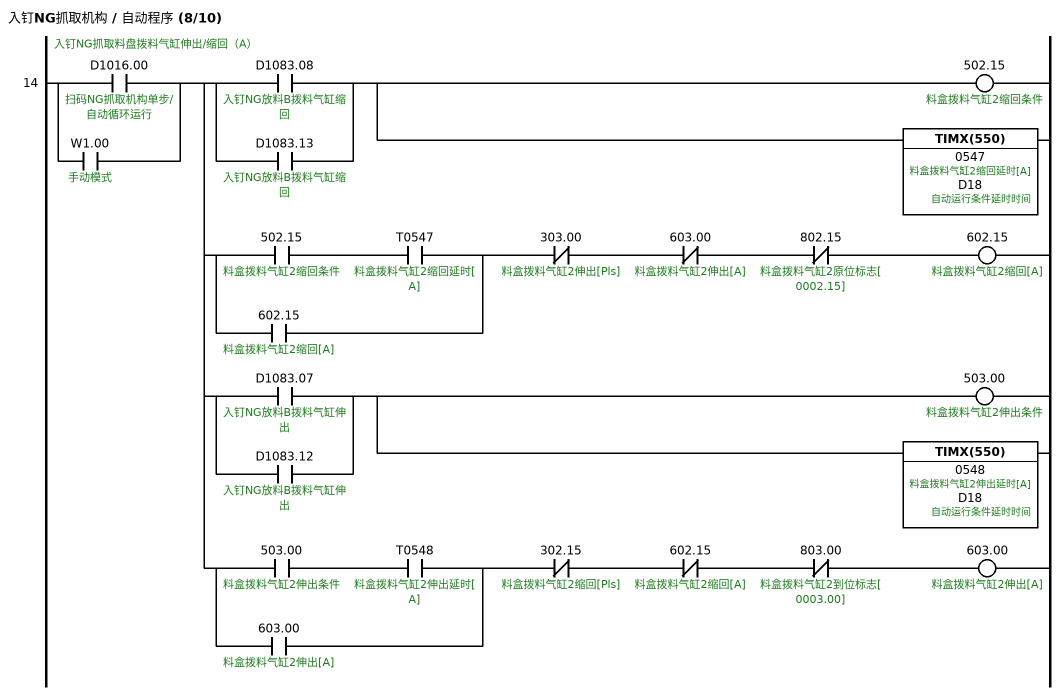
; [picture p144: 入钉NG抓取机构 / 自动程序, rungs 14-14]
; rung 14: 入钉NG抓取料盘拨料气缸伸出/缩回（A）
LD D1016.00  ; 扫码NG抓取机构单步/自动循环运行
OR W1.00  ; 手动模式
OUT TR0
LD D1083.08  ; 入钉NG放料B拨料气缸缩回
OR D1083.13  ; 入钉NG放料B拨料气缸缩回
ANDLD
OUT 502.15  ; 料盒拨料气缸2缩回条件
TIMX(550) 0547 D18  ; 自动运行条件延时时间, 料盒拨料气缸2缩回延时[A]
LD TR0
LD 502.15  ; 料盒拨料气缸2缩回条件
AND T0547  ; 料盒拨料气缸2缩回延时[A]
OR 602.15  ; 料盒拨料气缸2缩回[A]
ANDLD
ANDNOT 303.00  ; 料盒拨料气缸2伸出[Pls]
ANDNOT 603.00  ; 料盒拨料气缸2伸出[A]
ANDNOT 802.15  ; 料盒拨料气缸2原位标志[0002.15]
OUT 602.15  ; 料盒拨料气缸2缩回[A]
LD TR0
LD D1083.07  ; 入钉NG放料B拨料气缸伸出
OR D1083.12  ; 入钉NG放料B拨料气缸伸出
ANDLD
OUT 503.00  ; 料盒拨料气缸2伸出条件
TIMX(550) 0548 D18  ; 自动运行条件延时时间, 料盒拨料气缸2伸出延时[A]
LD TR0
LD 503.00  ; 料盒拨料气缸2伸出条件
AND T0548  ; 料盒拨料气缸2伸出延时[A]
OR 603.00  ; 料盒拨料气缸2伸出[A]
ANDLD
ANDNOT 302.15  ; 料盒拨料气缸2缩回[Pls]
ANDNOT 602.15  ; 料盒拨料气缸2缩回[A]
ANDNOT 803.00  ; 料盒拨料气缸2到位标志[0003.00]
OUT 603.00  ; 料盒拨料气缸2伸出[A]

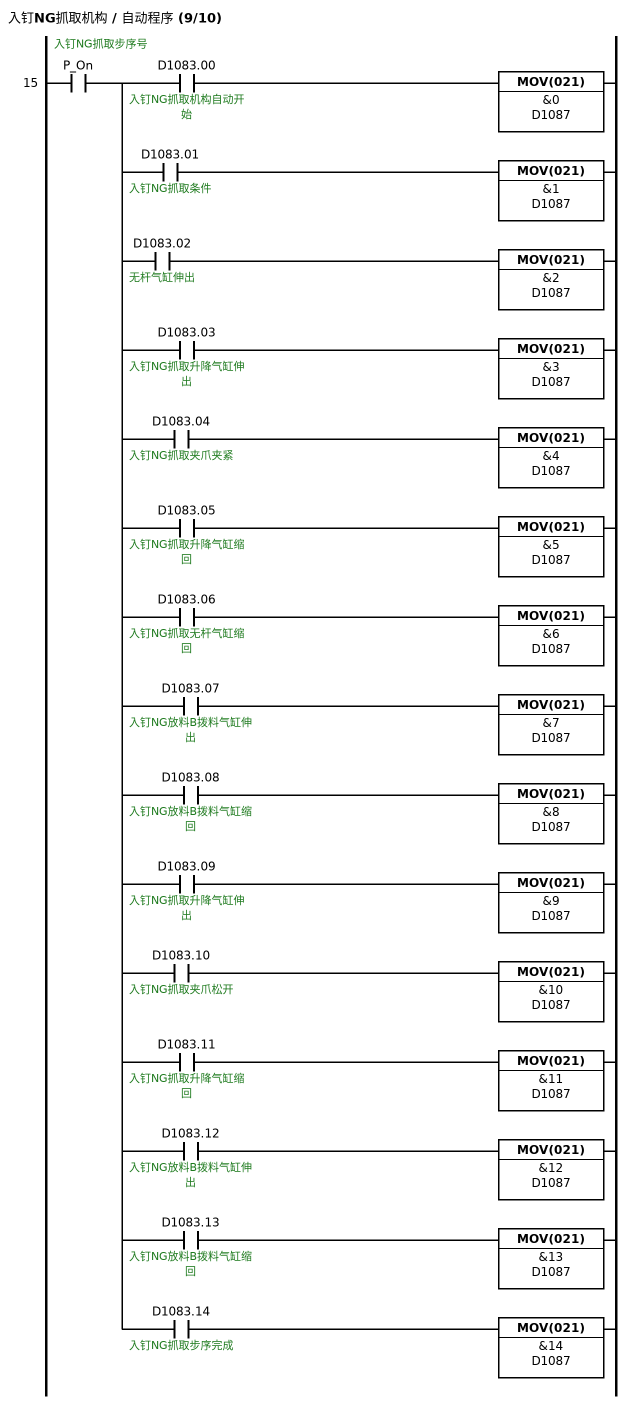
; rung 15: 入钉NG抓取步序号
LD P_On
OUT TR0
AND D1083.00  ; 入钉NG抓取机构自动开始
MOV(021) &0 D1087
LD TR0
AND D1083.01  ; 入钉NG抓取条件
MOV(021) &1 D1087
LD TR0
AND D1083.02  ; 无杆气缸伸出
MOV(021) &2 D1087
LD TR0
AND D1083.03  ; 入钉NG抓取升降气缸伸出
MOV(021) &3 D1087
LD TR0
AND D1083.04  ; 入钉NG抓取夹爪夹紧
MOV(021) &4 D1087
LD TR0
AND D1083.05  ; 入钉NG抓取升降气缸缩回
MOV(021) &5 D1087
LD TR0
AND D1083.06  ; 入钉NG抓取无杆气缸缩回
MOV(021) &6 D1087
LD TR0
AND D1083.07  ; 入钉NG放料B拨料气缸伸出
MOV(021) &7 D1087
LD TR0
AND D1083.08  ; 入钉NG放料B拨料气缸缩回
MOV(021) &8 D1087
LD TR0
AND D1083.09  ; 入钉NG抓取升降气缸伸出
MOV(021) &9 D1087
LD TR0
AND D1083.10  ; 入钉NG抓取夹爪松开
MOV(021) &10 D1087
LD TR0
AND D1083.11  ; 入钉NG抓取升降气缸缩回
MOV(021) &11 D1087
LD TR0
AND D1083.12  ; 入钉NG放料B拨料气缸伸出
MOV(021) &12 D1087
LD TR0
AND D1083.13  ; 入钉NG放料B拨料气缸缩回
MOV(021) &13 D1087
LD TR0
AND D1083.14  ; 入钉NG抓取步序完成
MOV(021) &14 D1087

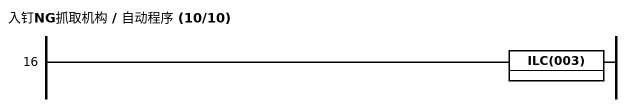
; rung 16
ILC(003)

### Section 状态指示灯

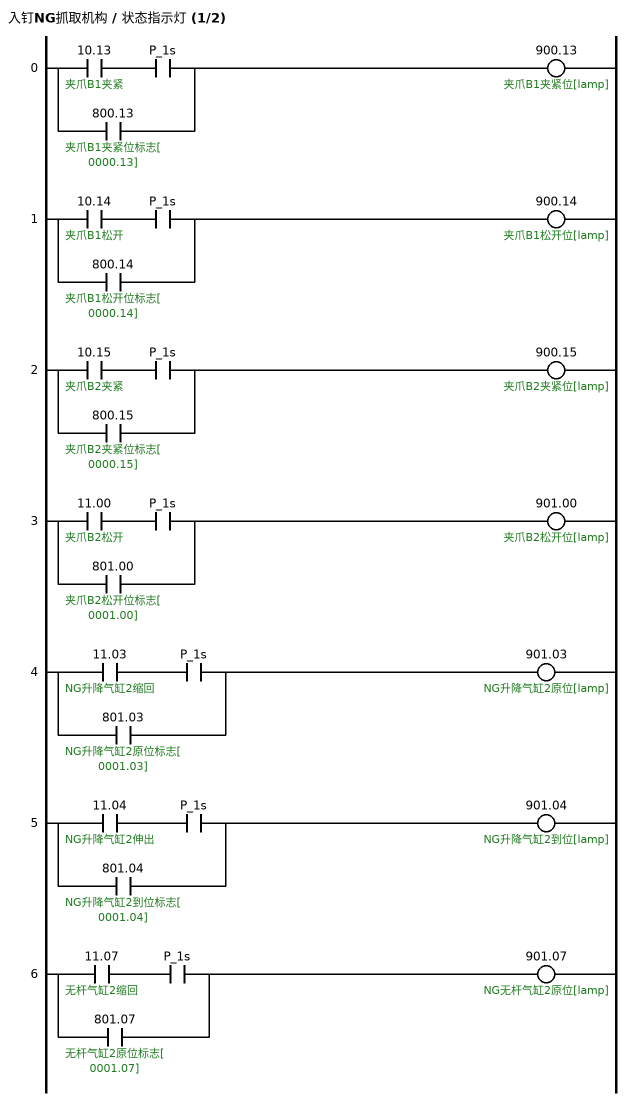
; rung 0
LD 10.13  ; 夹爪B1夹紧
AND P_1s
OR 800.13  ; 夹爪B1夹紧位标志[0000.13]
OUT 900.13  ; 夹爪B1夹紧位[lamp]
; rung 1
LD 10.14  ; 夹爪B1松开
AND P_1s
OR 800.14  ; 夹爪B1松开位标志[0000.14]
OUT 900.14  ; 夹爪B1松开位[lamp]
; rung 2
LD 10.15  ; 夹爪B2夹紧
AND P_1s
OR 800.15  ; 夹爪B2夹紧位标志[0000.15]
OUT 900.15  ; 夹爪B2夹紧位[lamp]
; rung 3
LD 11.00  ; 夹爪B2松开
AND P_1s
OR 801.00  ; 夹爪B2松开位标志[0001.00]
OUT 901.00  ; 夹爪B2松开位[lamp]
; rung 4
LD 11.03  ; NG升降气缸2缩回
AND P_1s
OR 801.03  ; NG升降气缸2原位标志[0001.03]
OUT 901.03  ; NG升降气缸2原位[lamp]
; rung 5
LD 11.04  ; NG升降气缸2伸出
AND P_1s
OR 801.04  ; NG升降气缸2到位标志[0001.04]
OUT 901.04  ; NG升降气缸2到位[lamp]
; rung 6
LD 11.07  ; 无杆气缸2缩回
AND P_1s
OR 801.07  ; 无杆气缸2原位标志[0001.07]
OUT 901.07  ; NG无杆气缸2原位[lamp]

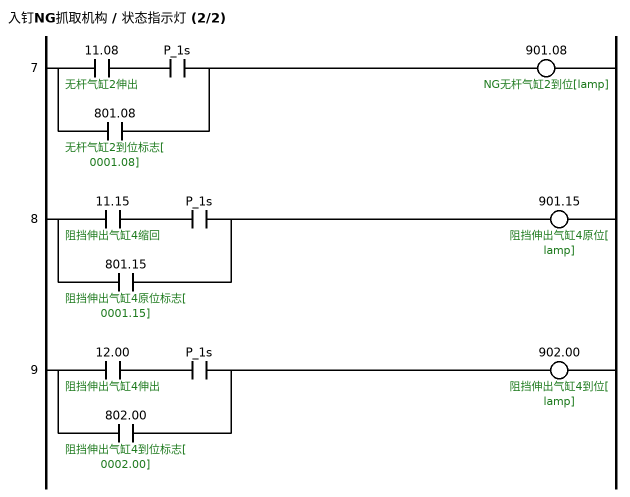
; rung 7
LD 11.08  ; 无杆气缸2伸出
AND P_1s
OR 801.08  ; 无杆气缸2到位标志[0001.08]
OUT 901.08  ; NG无杆气缸2到位[lamp]
; rung 8
LD 11.15  ; 阻挡伸出气缸4缩回
AND P_1s
OR 801.15  ; 阻挡伸出气缸4原位标志[0001.15]
OUT 901.15  ; 阻挡伸出气缸4原位[lamp]
; rung 9
LD 12.00  ; 阻挡伸出气缸4伸出
AND P_1s
OR 802.00  ; 阻挡伸出气缸4到位标志[0002.00]
OUT 902.00  ; 阻挡伸出气缸4到位[lamp]

### Section 输出程序

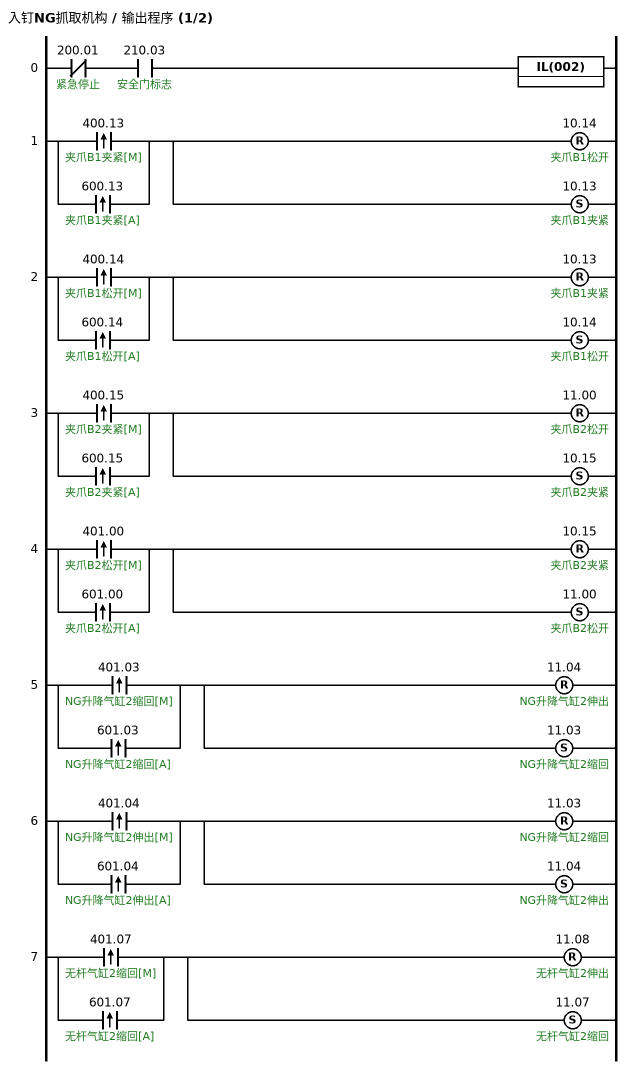
; rung 0
LDNOT 200.01  ; 紧急停止
AND 210.03  ; 安全门标志
IL(002)
; rung 1
@LD 400.13  ; 夹爪B1夹紧[M]
@OR 600.13  ; 夹爪B1夹紧[A]
RSET 10.14  ; 夹爪B1松开
SET 10.13  ; 夹爪B1夹紧
; rung 2
@LD 400.14  ; 夹爪B1松开[M]
@OR 600.14  ; 夹爪B1松开[A]
RSET 10.13  ; 夹爪B1夹紧
SET 10.14  ; 夹爪B1松开
; rung 3
@LD 400.15  ; 夹爪B2夹紧[M]
@OR 600.15  ; 夹爪B2夹紧[A]
RSET 11.00  ; 夹爪B2松开
SET 10.15  ; 夹爪B2夹紧
; rung 4
@LD 401.00  ; 夹爪B2松开[M]
@OR 601.00  ; 夹爪B2松开[A]
RSET 10.15  ; 夹爪B2夹紧
SET 11.00  ; 夹爪B2松开
; rung 5
@LD 401.03  ; NG升降气缸2缩回[M]
@OR 601.03  ; NG升降气缸2缩回[A]
RSET 11.04  ; NG升降气缸2伸出
SET 11.03  ; NG升降气缸2缩回
; rung 6
@LD 401.04  ; NG升降气缸2伸出[M]
@OR 601.04  ; NG升降气缸2伸出[A]
RSET 11.03  ; NG升降气缸2缩回
SET 11.04  ; NG升降气缸2伸出
; rung 7
@LD 401.07  ; 无杆气缸2缩回[M]
@OR 601.07  ; 无杆气缸2缩回[A]
RSET 11.08  ; 无杆气缸2伸出
SET 11.07  ; 无杆气缸2缩回

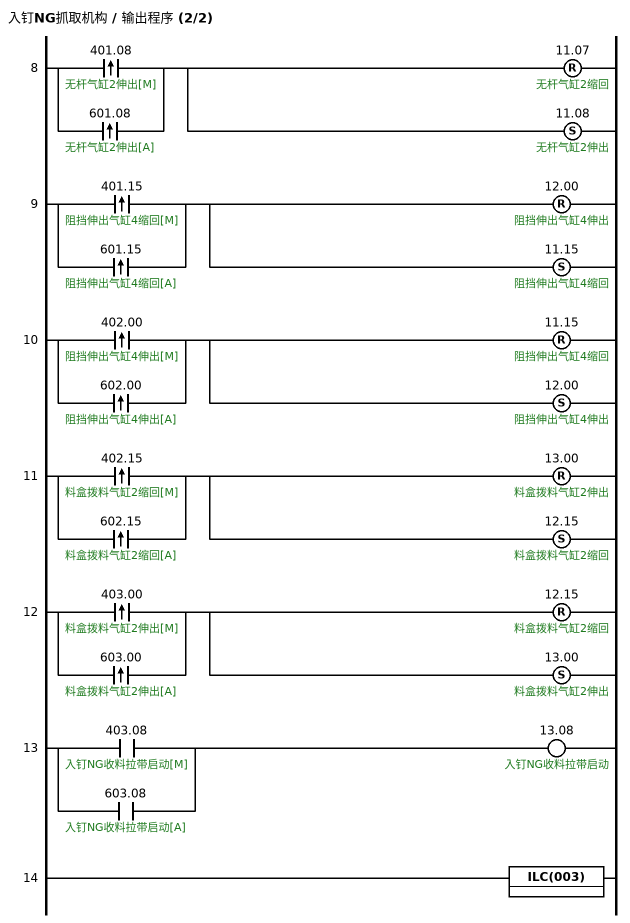
; rung 8
@LD 401.08  ; 无杆气缸2伸出[M]
@OR 601.08  ; 无杆气缸2伸出[A]
RSET 11.07  ; 无杆气缸2缩回
SET 11.08  ; 无杆气缸2伸出
; rung 9
@LD 401.15  ; 阻挡伸出气缸4缩回[M]
@OR 601.15  ; 阻挡伸出气缸4缩回[A]
RSET 12.00  ; 阻挡伸出气缸4伸出
SET 11.15  ; 阻挡伸出气缸4缩回
; rung 10
@LD 402.00  ; 阻挡伸出气缸4伸出[M]
@OR 602.00  ; 阻挡伸出气缸4伸出[A]
RSET 11.15  ; 阻挡伸出气缸4缩回
SET 12.00  ; 阻挡伸出气缸4伸出
; rung 11
@LD 402.15  ; 料盒拨料气缸2缩回[M]
@OR 602.15  ; 料盒拨料气缸2缩回[A]
RSET 13.00  ; 料盒拨料气缸2伸出
SET 12.15  ; 料盒拨料气缸2缩回
; rung 12
@LD 403.00  ; 料盒拨料气缸2伸出[M]
@OR 603.00  ; 料盒拨料气缸2伸出[A]
RSET 12.15  ; 料盒拨料气缸2缩回
SET 13.00  ; 料盒拨料气缸2伸出
; rung 13
LD 403.08  ; 入钉NG收料拉带启动[M]
OR 603.08  ; 入钉NG收料拉带启动[A]
OUT 13.08  ; 入钉NG收料拉带启动
; rung 14
ILC(003)

### Section END
; rung 0
END(001)

## Program COMMON (cyclic task 6)

### Section 传感器延时

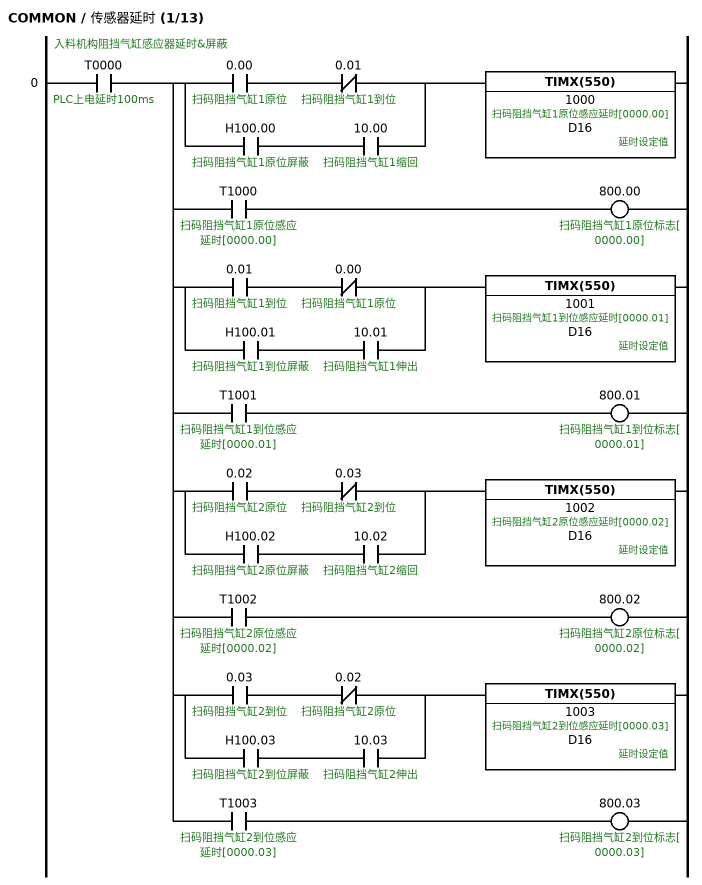
; rung 0: 入料机构阻挡气缸感应器延时&屏蔽
LD T0000  ; PLC上电延时100ms
OUT TR0
LD 0.00  ; 扫码阻挡气缸1原位
ANDNOT 0.01  ; 扫码阻挡气缸1到位
LD H100.00  ; 扫码阻挡气缸1原位屏蔽
AND 10.00  ; 扫码阻挡气缸1缩回
ORLD
ANDLD
TIMX(550) 1000 D16  ; 延时设定值, 扫码阻挡气缸1原位感应延时[0000.00]
LD TR0
AND T1000  ; 扫码阻挡气缸1原位感应延时[0000.00]
OUT 800.00  ; 扫码阻挡气缸1原位标志[0000.00]
LD TR0
LD 0.01  ; 扫码阻挡气缸1到位
ANDNOT 0.00  ; 扫码阻挡气缸1原位
LD H100.01  ; 扫码阻挡气缸1到位屏蔽
AND 10.01  ; 扫码阻挡气缸1伸出
ORLD
ANDLD
TIMX(550) 1001 D16  ; 延时设定值, 扫码阻挡气缸1到位感应延时[0000.01]
LD TR0
AND T1001  ; 扫码阻挡气缸1到位感应延时[0000.01]
OUT 800.01  ; 扫码阻挡气缸1到位标志[0000.01]
LD TR0
LD 0.02  ; 扫码阻挡气缸2原位
ANDNOT 0.03  ; 扫码阻挡气缸2到位
LD H100.02  ; 扫码阻挡气缸2原位屏蔽
AND 10.02  ; 扫码阻挡气缸2缩回
ORLD
ANDLD
TIMX(550) 1002 D16  ; 延时设定值, 扫码阻挡气缸2原位感应延时[0000.02]
LD TR0
AND T1002  ; 扫码阻挡气缸2原位感应延时[0000.02]
OUT 800.02  ; 扫码阻挡气缸2原位标志[0000.02]
LD TR0
LD 0.03  ; 扫码阻挡气缸2到位
ANDNOT 0.02  ; 扫码阻挡气缸2原位
LD H100.03  ; 扫码阻挡气缸2到位屏蔽
AND 10.03  ; 扫码阻挡气缸2伸出
ORLD
ANDLD
TIMX(550) 1003 D16  ; 延时设定值, 扫码阻挡气缸2到位感应延时[0000.03]
LD TR0
AND T1003  ; 扫码阻挡气缸2到位感应延时[0000.03]
OUT 800.03  ; 扫码阻挡气缸2到位标志[0000.03]

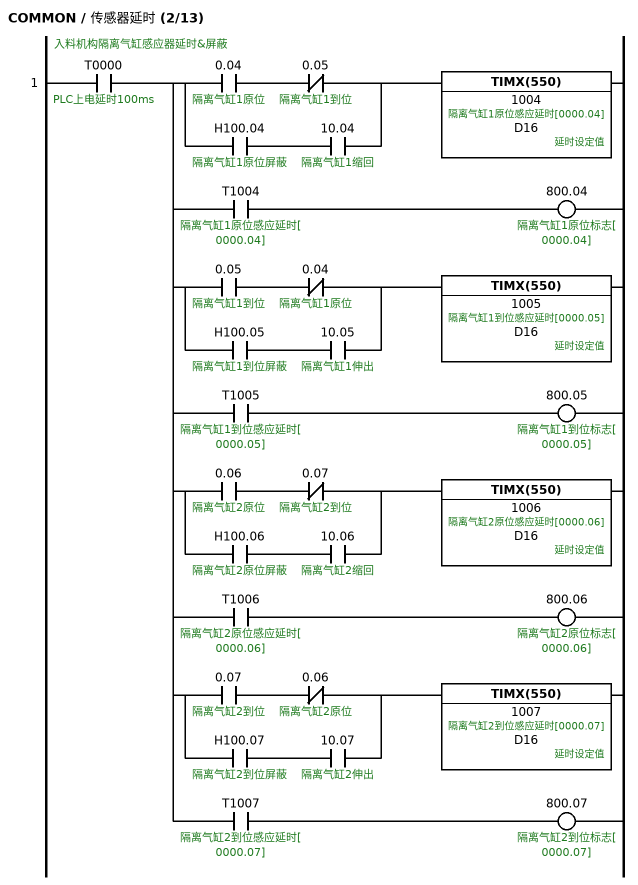
; rung 1: 入料机构隔离气缸感应器延时&屏蔽
LD T0000  ; PLC上电延时100ms
OUT TR0
LD 0.04  ; 隔离气缸1原位
ANDNOT 0.05  ; 隔离气缸1到位
LD H100.04  ; 隔离气缸1原位屏蔽
AND 10.04  ; 隔离气缸1缩回
ORLD
ANDLD
TIMX(550) 1004 D16  ; 延时设定值, 隔离气缸1原位感应延时[0000.04]
LD TR0
AND T1004  ; 隔离气缸1原位感应延时[0000.04]
OUT 800.04  ; 隔离气缸1原位标志[0000.04]
LD TR0
LD 0.05  ; 隔离气缸1到位
ANDNOT 0.04  ; 隔离气缸1原位
LD H100.05  ; 隔离气缸1到位屏蔽
AND 10.05  ; 隔离气缸1伸出
ORLD
ANDLD
TIMX(550) 1005 D16  ; 延时设定值, 隔离气缸1到位感应延时[0000.05]
LD TR0
AND T1005  ; 隔离气缸1到位感应延时[0000.05]
OUT 800.05  ; 隔离气缸1到位标志[0000.05]
LD TR0
LD 0.06  ; 隔离气缸2原位
ANDNOT 0.07  ; 隔离气缸2到位
LD H100.06  ; 隔离气缸2原位屏蔽
AND 10.06  ; 隔离气缸2缩回
ORLD
ANDLD
TIMX(550) 1006 D16  ; 延时设定值, 隔离气缸2原位感应延时[0000.06]
LD TR0
AND T1006  ; 隔离气缸2原位感应延时[0000.06]
OUT 800.06  ; 隔离气缸2原位标志[0000.06]
LD TR0
LD 0.07  ; 隔离气缸2到位
ANDNOT 0.06  ; 隔离气缸2原位
LD H100.07  ; 隔离气缸2到位屏蔽
AND 10.07  ; 隔离气缸2伸出
ORLD
ANDLD
TIMX(550) 1007 D16  ; 延时设定值, 隔离气缸2到位感应延时[0000.07]
LD TR0
AND T1007  ; 隔离气缸2到位感应延时[0000.07]
OUT 800.07  ; 隔离气缸2到位标志[0000.07]

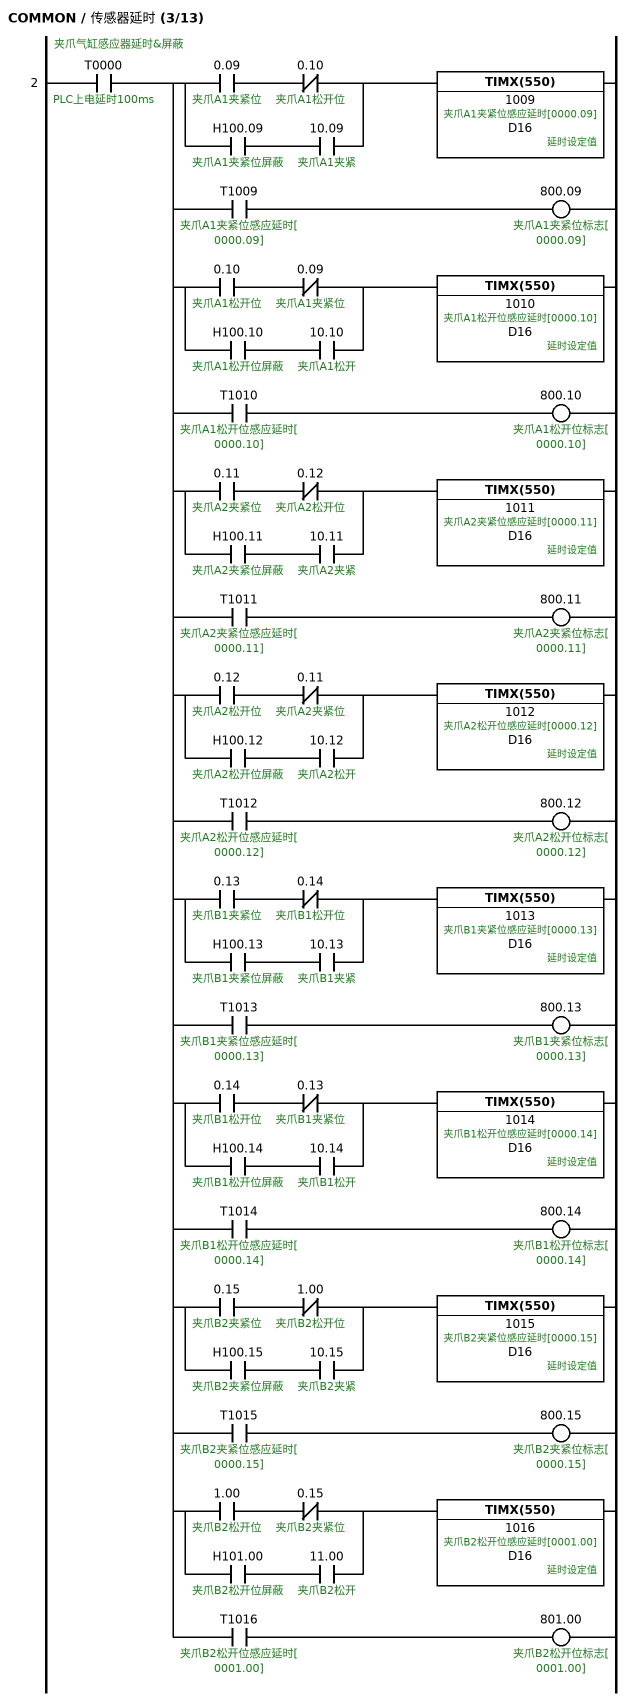
; rung 2: 夹爪气缸感应器延时&屏蔽
LD T0000  ; PLC上电延时100ms
OUT TR0
LD 0.09  ; 夹爪A1夹紧位
ANDNOT 0.10  ; 夹爪A1松开位
LD H100.09  ; 夹爪A1夹紧位屏蔽
AND 10.09  ; 夹爪A1夹紧
ORLD
ANDLD
TIMX(550) 1009 D16  ; 延时设定值, 夹爪A1夹紧位感应延时[0000.09]
LD TR0
AND T1009  ; 夹爪A1夹紧位感应延时[0000.09]
OUT 800.09  ; 夹爪A1夹紧位标志[0000.09]
LD TR0
LD 0.10  ; 夹爪A1松开位
ANDNOT 0.09  ; 夹爪A1夹紧位
LD H100.10  ; 夹爪A1松开位屏蔽
AND 10.10  ; 夹爪A1松开
ORLD
ANDLD
TIMX(550) 1010 D16  ; 延时设定值, 夹爪A1松开位感应延时[0000.10]
LD TR0
AND T1010  ; 夹爪A1松开位感应延时[0000.10]
OUT 800.10  ; 夹爪A1松开位标志[0000.10]
LD TR0
LD 0.11  ; 夹爪A2夹紧位
ANDNOT 0.12  ; 夹爪A2松开位
LD H100.11  ; 夹爪A2夹紧位屏蔽
AND 10.11  ; 夹爪A2夹紧
ORLD
ANDLD
TIMX(550) 1011 D16  ; 延时设定值, 夹爪A2夹紧位感应延时[0000.11]
LD TR0
AND T1011  ; 夹爪A2夹紧位感应延时[0000.11]
OUT 800.11  ; 夹爪A2夹紧位标志[0000.11]
LD TR0
LD 0.12  ; 夹爪A2松开位
ANDNOT 0.11  ; 夹爪A2夹紧位
LD H100.12  ; 夹爪A2松开位屏蔽
AND 10.12  ; 夹爪A2松开
ORLD
ANDLD
TIMX(550) 1012 D16  ; 延时设定值, 夹爪A2松开位感应延时[0000.12]
LD TR0
AND T1012  ; 夹爪A2松开位感应延时[0000.12]
OUT 800.12  ; 夹爪A2松开位标志[0000.12]
LD TR0
LD 0.13  ; 夹爪B1夹紧位
ANDNOT 0.14  ; 夹爪B1松开位
LD H100.13  ; 夹爪B1夹紧位屏蔽
AND 10.13  ; 夹爪B1夹紧
ORLD
ANDLD
TIMX(550) 1013 D16  ; 延时设定值, 夹爪B1夹紧位感应延时[0000.13]
LD TR0
AND T1013  ; 夹爪B1夹紧位感应延时[0000.13]
OUT 800.13  ; 夹爪B1夹紧位标志[0000.13]
LD TR0
LD 0.14  ; 夹爪B1松开位
ANDNOT 0.13  ; 夹爪B1夹紧位
LD H100.14  ; 夹爪B1松开位屏蔽
AND 10.14  ; 夹爪B1松开
ORLD
ANDLD
TIMX(550) 1014 D16  ; 延时设定值, 夹爪B1松开位感应延时[0000.14]
LD TR0
AND T1014  ; 夹爪B1松开位感应延时[0000.14]
OUT 800.14  ; 夹爪B1松开位标志[0000.14]
LD TR0
LD 0.15  ; 夹爪B2夹紧位
ANDNOT 1.00  ; 夹爪B2松开位
LD H100.15  ; 夹爪B2夹紧位屏蔽
AND 10.15  ; 夹爪B2夹紧
ORLD
ANDLD
TIMX(550) 1015 D16  ; 延时设定值, 夹爪B2夹紧位感应延时[0000.15]
LD TR0
AND T1015  ; 夹爪B2夹紧位感应延时[0000.15]
OUT 800.15  ; 夹爪B2夹紧位标志[0000.15]
LD TR0
LD 1.00  ; 夹爪B2松开位
ANDNOT 0.15  ; 夹爪B2夹紧位
LD H101.00  ; 夹爪B2松开位屏蔽
AND 11.00  ; 夹爪B2松开
ORLD
ANDLD
TIMX(550) 1016 D16  ; 延时设定值, 夹爪B2松开位感应延时[0001.00]
LD TR0
AND T1016  ; 夹爪B2松开位感应延时[0001.00]
OUT 801.00  ; 夹爪B2松开位标志[0001.00]

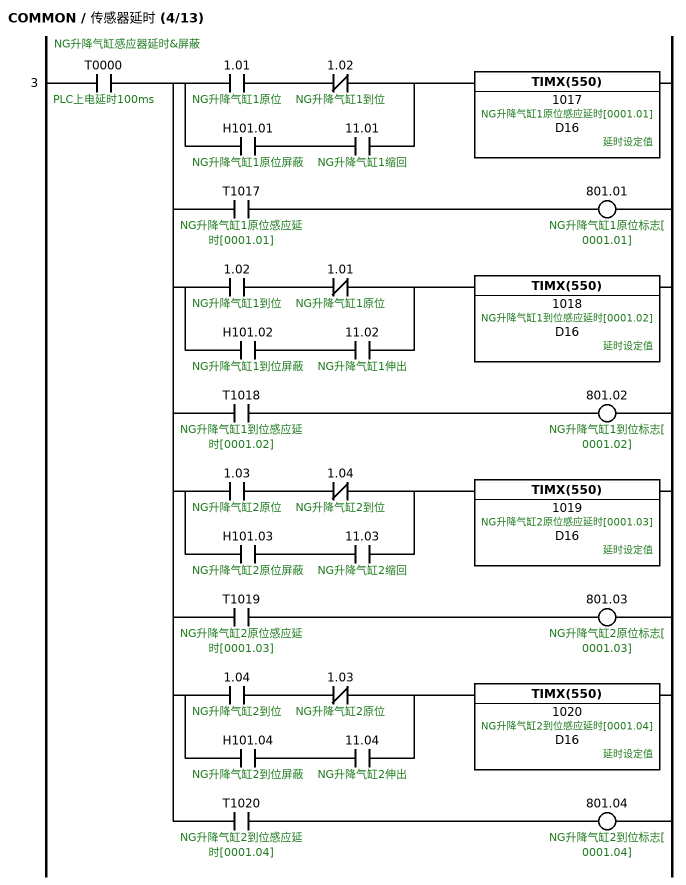
; rung 3: NG升降气缸感应器延时&屏蔽
LD T0000  ; PLC上电延时100ms
OUT TR0
LD 1.01  ; NG升降气缸1原位
ANDNOT 1.02  ; NG升降气缸1到位
LD H101.01  ; NG升降气缸1原位屏蔽
AND 11.01  ; NG升降气缸1缩回
ORLD
ANDLD
TIMX(550) 1017 D16  ; 延时设定值, NG升降气缸1原位感应延时[0001.01]
LD TR0
AND T1017  ; NG升降气缸1原位感应延时[0001.01]
OUT 801.01  ; NG升降气缸1原位标志[0001.01]
LD TR0
LD 1.02  ; NG升降气缸1到位
ANDNOT 1.01  ; NG升降气缸1原位
LD H101.02  ; NG升降气缸1到位屏蔽
AND 11.02  ; NG升降气缸1伸出
ORLD
ANDLD
TIMX(550) 1018 D16  ; 延时设定值, NG升降气缸1到位感应延时[0001.02]
LD TR0
AND T1018  ; NG升降气缸1到位感应延时[0001.02]
OUT 801.02  ; NG升降气缸1到位标志[0001.02]
LD TR0
LD 1.03  ; NG升降气缸2原位
ANDNOT 1.04  ; NG升降气缸2到位
LD H101.03  ; NG升降气缸2原位屏蔽
AND 11.03  ; NG升降气缸2缩回
ORLD
ANDLD
TIMX(550) 1019 D16  ; 延时设定值, NG升降气缸2原位感应延时[0001.03]
LD TR0
AND T1019  ; NG升降气缸2原位感应延时[0001.03]
OUT 801.03  ; NG升降气缸2原位标志[0001.03]
LD TR0
LD 1.04  ; NG升降气缸2到位
ANDNOT 1.03  ; NG升降气缸2原位
LD H101.04  ; NG升降气缸2到位屏蔽
AND 11.04  ; NG升降气缸2伸出
ORLD
ANDLD
TIMX(550) 1020 D16  ; 延时设定值, NG升降气缸2到位感应延时[0001.04]
LD TR0
AND T1020  ; NG升降气缸2到位感应延时[0001.04]
OUT 801.04  ; NG升降气缸2到位标志[0001.04]

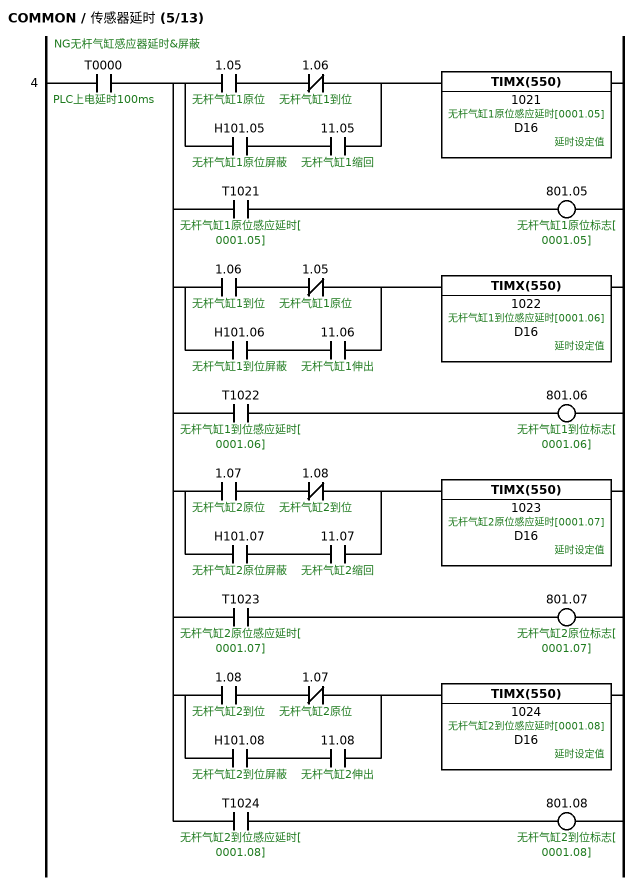
; rung 4: NG无杆气缸感应器延时&屏蔽
LD T0000  ; PLC上电延时100ms
OUT TR0
LD 1.05  ; 无杆气缸1原位
ANDNOT 1.06  ; 无杆气缸1到位
LD H101.05  ; 无杆气缸1原位屏蔽
AND 11.05  ; 无杆气缸1缩回
ORLD
ANDLD
TIMX(550) 1021 D16  ; 延时设定值, 无杆气缸1原位感应延时[0001.05]
LD TR0
AND T1021  ; 无杆气缸1原位感应延时[0001.05]
OUT 801.05  ; 无杆气缸1原位标志[0001.05]
LD TR0
LD 1.06  ; 无杆气缸1到位
ANDNOT 1.05  ; 无杆气缸1原位
LD H101.06  ; 无杆气缸1到位屏蔽
AND 11.06  ; 无杆气缸1伸出
ORLD
ANDLD
TIMX(550) 1022 D16  ; 延时设定值, 无杆气缸1到位感应延时[0001.06]
LD TR0
AND T1022  ; 无杆气缸1到位感应延时[0001.06]
OUT 801.06  ; 无杆气缸1到位标志[0001.06]
LD TR0
LD 1.07  ; 无杆气缸2原位
ANDNOT 1.08  ; 无杆气缸2到位
LD H101.07  ; 无杆气缸2原位屏蔽
AND 11.07  ; 无杆气缸2缩回
ORLD
ANDLD
TIMX(550) 1023 D16  ; 延时设定值, 无杆气缸2原位感应延时[0001.07]
LD TR0
AND T1023  ; 无杆气缸2原位感应延时[0001.07]
OUT 801.07  ; 无杆气缸2原位标志[0001.07]
LD TR0
LD 1.08  ; 无杆气缸2到位
ANDNOT 1.07  ; 无杆气缸2原位
LD H101.08  ; 无杆气缸2到位屏蔽
AND 11.08  ; 无杆气缸2伸出
ORLD
ANDLD
TIMX(550) 1024 D16  ; 延时设定值, 无杆气缸2到位感应延时[0001.08]
LD TR0
AND T1024  ; 无杆气缸2到位感应延时[0001.08]
OUT 801.08  ; 无杆气缸2到位标志[0001.08]

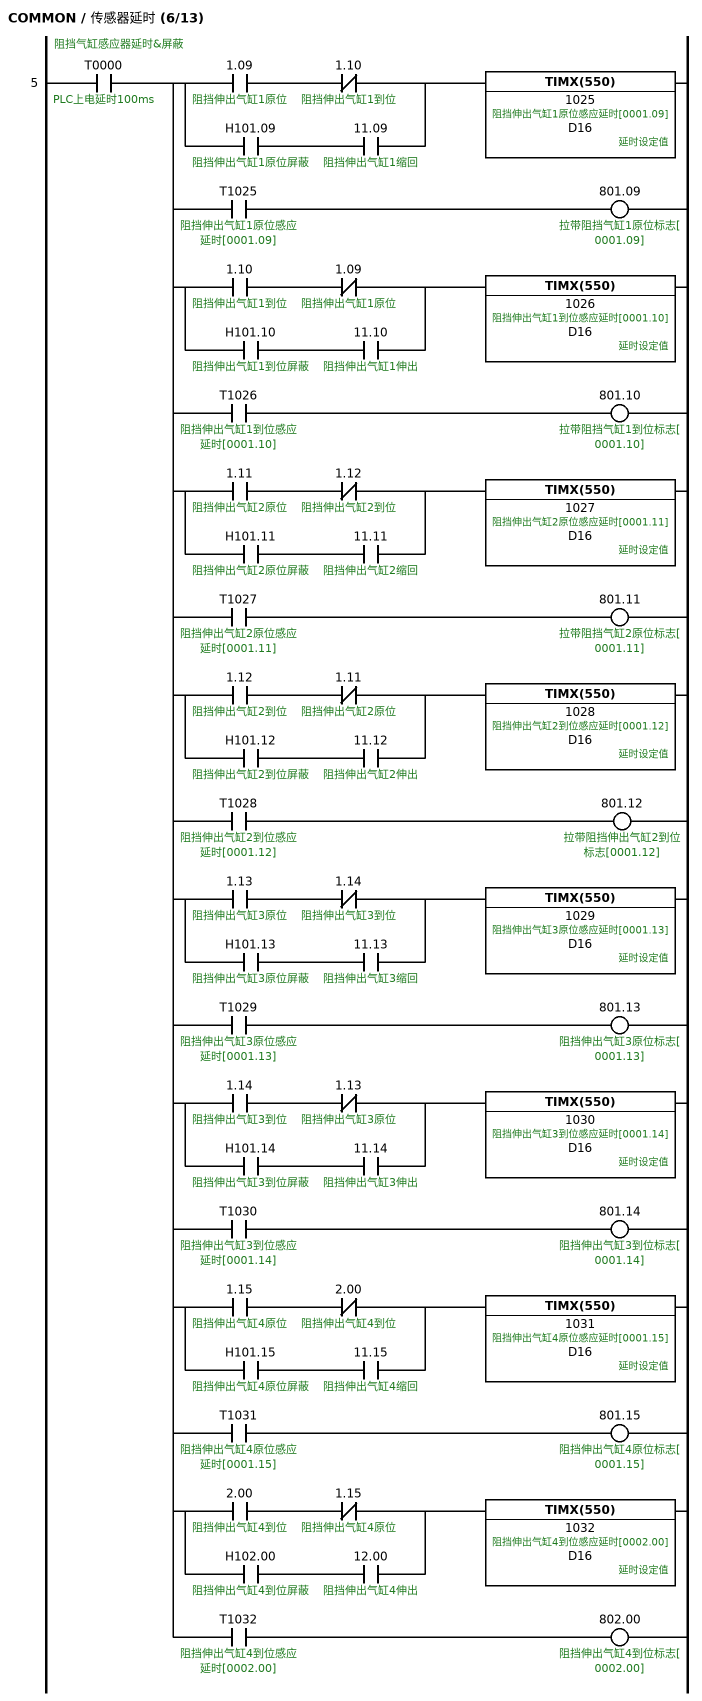
; rung 5: 阻挡气缸感应器延时&屏蔽
LD T0000  ; PLC上电延时100ms
OUT TR0
LD 1.09  ; 阻挡伸出气缸1原位
ANDNOT 1.10  ; 阻挡伸出气缸1到位
LD H101.09  ; 阻挡伸出气缸1原位屏蔽
AND 11.09  ; 阻挡伸出气缸1缩回
ORLD
ANDLD
TIMX(550) 1025 D16  ; 延时设定值, 阻挡伸出气缸1原位感应延时[0001.09]
LD TR0
AND T1025  ; 阻挡伸出气缸1原位感应延时[0001.09]
OUT 801.09  ; 拉带阻挡气缸1原位标志[0001.09]
LD TR0
LD 1.10  ; 阻挡伸出气缸1到位
ANDNOT 1.09  ; 阻挡伸出气缸1原位
LD H101.10  ; 阻挡伸出气缸1到位屏蔽
AND 11.10  ; 阻挡伸出气缸1伸出
ORLD
ANDLD
TIMX(550) 1026 D16  ; 延时设定值, 阻挡伸出气缸1到位感应延时[0001.10]
LD TR0
AND T1026  ; 阻挡伸出气缸1到位感应延时[0001.10]
OUT 801.10  ; 拉带阻挡气缸1到位标志[0001.10]
LD TR0
LD 1.11  ; 阻挡伸出气缸2原位
ANDNOT 1.12  ; 阻挡伸出气缸2到位
LD H101.11  ; 阻挡伸出气缸2原位屏蔽
AND 11.11  ; 阻挡伸出气缸2缩回
ORLD
ANDLD
TIMX(550) 1027 D16  ; 延时设定值, 阻挡伸出气缸2原位感应延时[0001.11]
LD TR0
AND T1027  ; 阻挡伸出气缸2原位感应延时[0001.11]
OUT 801.11  ; 拉带阻挡气缸2原位标志[0001.11]
LD TR0
LD 1.12  ; 阻挡伸出气缸2到位
ANDNOT 1.11  ; 阻挡伸出气缸2原位
LD H101.12  ; 阻挡伸出气缸2到位屏蔽
AND 11.12  ; 阻挡伸出气缸2伸出
ORLD
ANDLD
TIMX(550) 1028 D16  ; 延时设定值, 阻挡伸出气缸2到位感应延时[0001.12]
LD TR0
AND T1028  ; 阻挡伸出气缸2到位感应延时[0001.12]
OUT 801.12  ; 拉带阻挡伸出气缸2到位标志[0001.12]
LD TR0
LD 1.13  ; 阻挡伸出气缸3原位
ANDNOT 1.14  ; 阻挡伸出气缸3到位
LD H101.13  ; 阻挡伸出气缸3原位屏蔽
AND 11.13  ; 阻挡伸出气缸3缩回
ORLD
ANDLD
TIMX(550) 1029 D16  ; 延时设定值, 阻挡伸出气缸3原位感应延时[0001.13]
LD TR0
AND T1029  ; 阻挡伸出气缸3原位感应延时[0001.13]
OUT 801.13  ; 阻挡伸出气缸3原位标志[0001.13]
LD TR0
LD 1.14  ; 阻挡伸出气缸3到位
ANDNOT 1.13  ; 阻挡伸出气缸3原位
LD H101.14  ; 阻挡伸出气缸3到位屏蔽
AND 11.14  ; 阻挡伸出气缸3伸出
ORLD
ANDLD
TIMX(550) 1030 D16  ; 延时设定值, 阻挡伸出气缸3到位感应延时[0001.14]
LD TR0
AND T1030  ; 阻挡伸出气缸3到位感应延时[0001.14]
OUT 801.14  ; 阻挡伸出气缸3到位标志[0001.14]
LD TR0
LD 1.15  ; 阻挡伸出气缸4原位
ANDNOT 2.00  ; 阻挡伸出气缸4到位
LD H101.15  ; 阻挡伸出气缸4原位屏蔽
AND 11.15  ; 阻挡伸出气缸4缩回
ORLD
ANDLD
TIMX(550) 1031 D16  ; 延时设定值, 阻挡伸出气缸4原位感应延时[0001.15]
LD TR0
AND T1031  ; 阻挡伸出气缸4原位感应延时[0001.15]
OUT 801.15  ; 阻挡伸出气缸4原位标志[0001.15]
LD TR0
LD 2.00  ; 阻挡伸出气缸4到位
ANDNOT 1.15  ; 阻挡伸出气缸4原位
LD H102.00  ; 阻挡伸出气缸4到位屏蔽
AND 12.00  ; 阻挡伸出气缸4伸出
ORLD
ANDLD
TIMX(550) 1032 D16  ; 延时设定值, 阻挡伸出气缸4到位感应延时[0002.00]
LD TR0
AND T1032  ; 阻挡伸出气缸4到位感应延时[0002.00]
OUT 802.00  ; 阻挡伸出气缸4到位标志[0002.00]

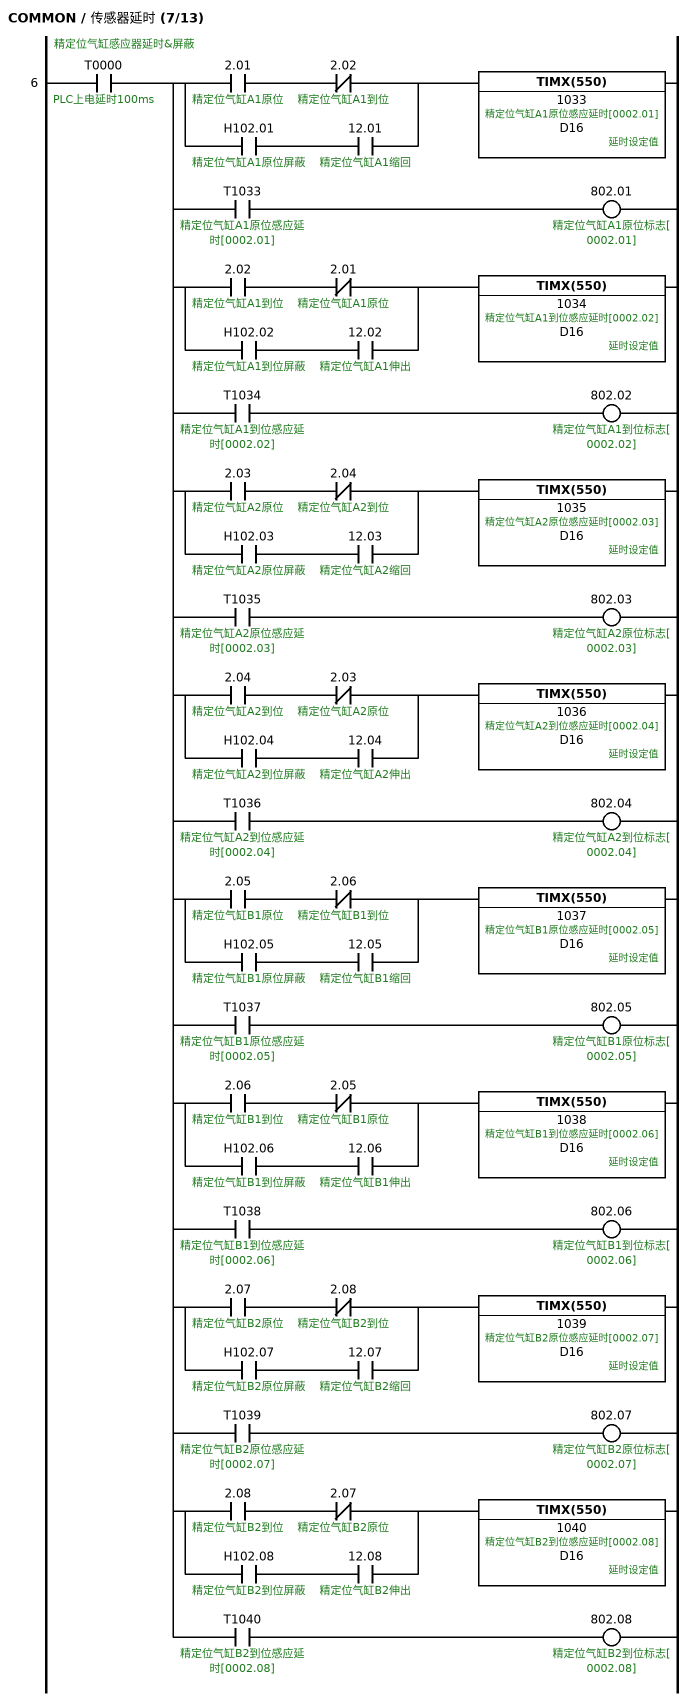
; rung 6: 精定位气缸感应器延时&屏蔽
LD T0000  ; PLC上电延时100ms
OUT TR0
LD 2.01  ; 精定位气缸A1原位
ANDNOT 2.02  ; 精定位气缸A1到位
LD H102.01  ; 精定位气缸A1原位屏蔽
AND 12.01  ; 精定位气缸A1缩回
ORLD
ANDLD
TIMX(550) 1033 D16  ; 延时设定值, 精定位气缸A1原位感应延时[0002.01]
LD TR0
AND T1033  ; 精定位气缸A1原位感应延时[0002.01]
OUT 802.01  ; 精定位气缸A1原位标志[0002.01]
LD TR0
LD 2.02  ; 精定位气缸A1到位
ANDNOT 2.01  ; 精定位气缸A1原位
LD H102.02  ; 精定位气缸A1到位屏蔽
AND 12.02  ; 精定位气缸A1伸出
ORLD
ANDLD
TIMX(550) 1034 D16  ; 延时设定值, 精定位气缸A1到位感应延时[0002.02]
LD TR0
AND T1034  ; 精定位气缸A1到位感应延时[0002.02]
OUT 802.02  ; 精定位气缸A1到位标志[0002.02]
LD TR0
LD 2.03  ; 精定位气缸A2原位
ANDNOT 2.04  ; 精定位气缸A2到位
LD H102.03  ; 精定位气缸A2原位屏蔽
AND 12.03  ; 精定位气缸A2缩回
ORLD
ANDLD
TIMX(550) 1035 D16  ; 延时设定值, 精定位气缸A2原位感应延时[0002.03]
LD TR0
AND T1035  ; 精定位气缸A2原位感应延时[0002.03]
OUT 802.03  ; 精定位气缸A2原位标志[0002.03]
LD TR0
LD 2.04  ; 精定位气缸A2到位
ANDNOT 2.03  ; 精定位气缸A2原位
LD H102.04  ; 精定位气缸A2到位屏蔽
AND 12.04  ; 精定位气缸A2伸出
ORLD
ANDLD
TIMX(550) 1036 D16  ; 延时设定值, 精定位气缸A2到位感应延时[0002.04]
LD TR0
AND T1036  ; 精定位气缸A2到位感应延时[0002.04]
OUT 802.04  ; 精定位气缸A2到位标志[0002.04]
LD TR0
LD 2.05  ; 精定位气缸B1原位
ANDNOT 2.06  ; 精定位气缸B1到位
LD H102.05  ; 精定位气缸B1原位屏蔽
AND 12.05  ; 精定位气缸B1缩回
ORLD
ANDLD
TIMX(550) 1037 D16  ; 延时设定值, 精定位气缸B1原位感应延时[0002.05]
LD TR0
AND T1037  ; 精定位气缸B1原位感应延时[0002.05]
OUT 802.05  ; 精定位气缸B1原位标志[0002.05]
LD TR0
LD 2.06  ; 精定位气缸B1到位
ANDNOT 2.05  ; 精定位气缸B1原位
LD H102.06  ; 精定位气缸B1到位屏蔽
AND 12.06  ; 精定位气缸B1伸出
ORLD
ANDLD
TIMX(550) 1038 D16  ; 延时设定值, 精定位气缸B1到位感应延时[0002.06]
LD TR0
AND T1038  ; 精定位气缸B1到位感应延时[0002.06]
OUT 802.06  ; 精定位气缸B1到位标志[0002.06]
LD TR0
LD 2.07  ; 精定位气缸B2原位
ANDNOT 2.08  ; 精定位气缸B2到位
LD H102.07  ; 精定位气缸B2原位屏蔽
AND 12.07  ; 精定位气缸B2缩回
ORLD
ANDLD
TIMX(550) 1039 D16  ; 延时设定值, 精定位气缸B2原位感应延时[0002.07]
LD TR0
AND T1039  ; 精定位气缸B2原位感应延时[0002.07]
OUT 802.07  ; 精定位气缸B2原位标志[0002.07]
LD TR0
LD 2.08  ; 精定位气缸B2到位
ANDNOT 2.07  ; 精定位气缸B2原位
LD H102.08  ; 精定位气缸B2到位屏蔽
AND 12.08  ; 精定位气缸B2伸出
ORLD
ANDLD
TIMX(550) 1040 D16  ; 延时设定值, 精定位气缸B2到位感应延时[0002.08]
LD TR0
AND T1040  ; 精定位气缸B2到位感应延时[0002.08]
OUT 802.08  ; 精定位气缸B2到位标志[0002.08]

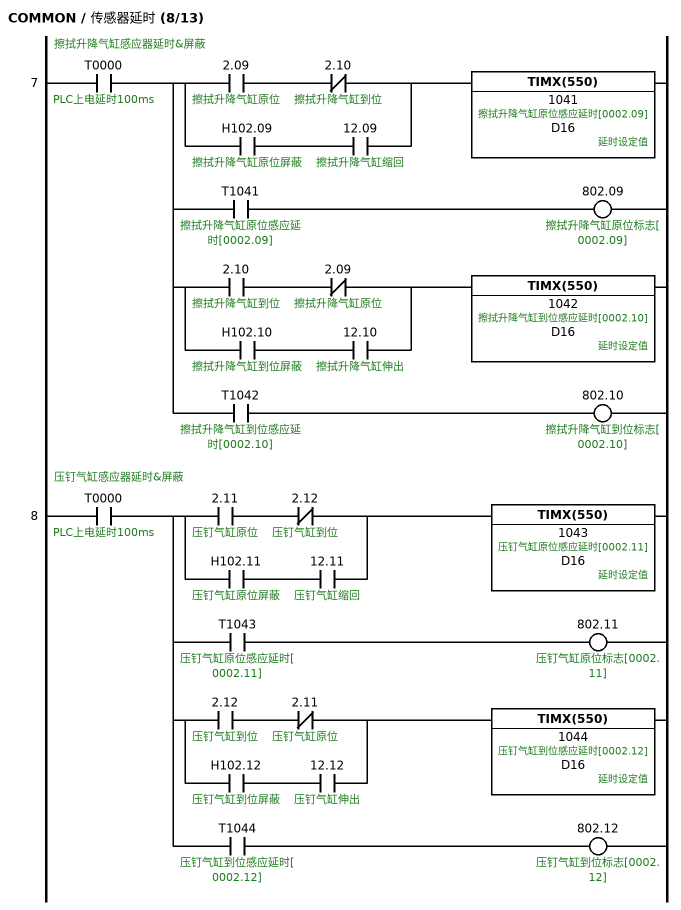
; rung 7: 擦拭升降气缸感应器延时&屏蔽
LD T0000  ; PLC上电延时100ms
OUT TR0
LD 2.09  ; 擦拭升降气缸原位
ANDNOT 2.10  ; 擦拭升降气缸到位
LD H102.09  ; 擦拭升降气缸原位屏蔽
AND 12.09  ; 擦拭升降气缸缩回
ORLD
ANDLD
TIMX(550) 1041 D16  ; 延时设定值, 擦拭升降气缸原位感应延时[0002.09]
LD TR0
AND T1041  ; 擦拭升降气缸原位感应延时[0002.09]
OUT 802.09  ; 擦拭升降气缸原位标志[0002.09]
LD TR0
LD 2.10  ; 擦拭升降气缸到位
ANDNOT 2.09  ; 擦拭升降气缸原位
LD H102.10  ; 擦拭升降气缸到位屏蔽
AND 12.10  ; 擦拭升降气缸伸出
ORLD
ANDLD
TIMX(550) 1042 D16  ; 延时设定值, 擦拭升降气缸到位感应延时[0002.10]
LD TR0
AND T1042  ; 擦拭升降气缸到位感应延时[0002.10]
OUT 802.10  ; 擦拭升降气缸到位标志[0002.10]
; rung 8: 压钉气缸感应器延时&屏蔽
LD T0000  ; PLC上电延时100ms
OUT TR0
LD 2.11  ; 压钉气缸原位
ANDNOT 2.12  ; 压钉气缸到位
LD H102.11  ; 压钉气缸原位屏蔽
AND 12.11  ; 压钉气缸缩回
ORLD
ANDLD
TIMX(550) 1043 D16  ; 延时设定值, 压钉气缸原位感应延时[0002.11]
LD TR0
AND T1043  ; 压钉气缸原位感应延时[0002.11]
OUT 802.11  ; 压钉气缸原位标志[0002.11]
LD TR0
LD 2.12  ; 压钉气缸到位
ANDNOT 2.11  ; 压钉气缸原位
LD H102.12  ; 压钉气缸到位屏蔽
AND 12.12  ; 压钉气缸伸出
ORLD
ANDLD
TIMX(550) 1044 D16  ; 延时设定值, 压钉气缸到位感应延时[0002.12]
LD TR0
AND T1044  ; 压钉气缸到位感应延时[0002.12]
OUT 802.12  ; 压钉气缸到位标志[0002.12]

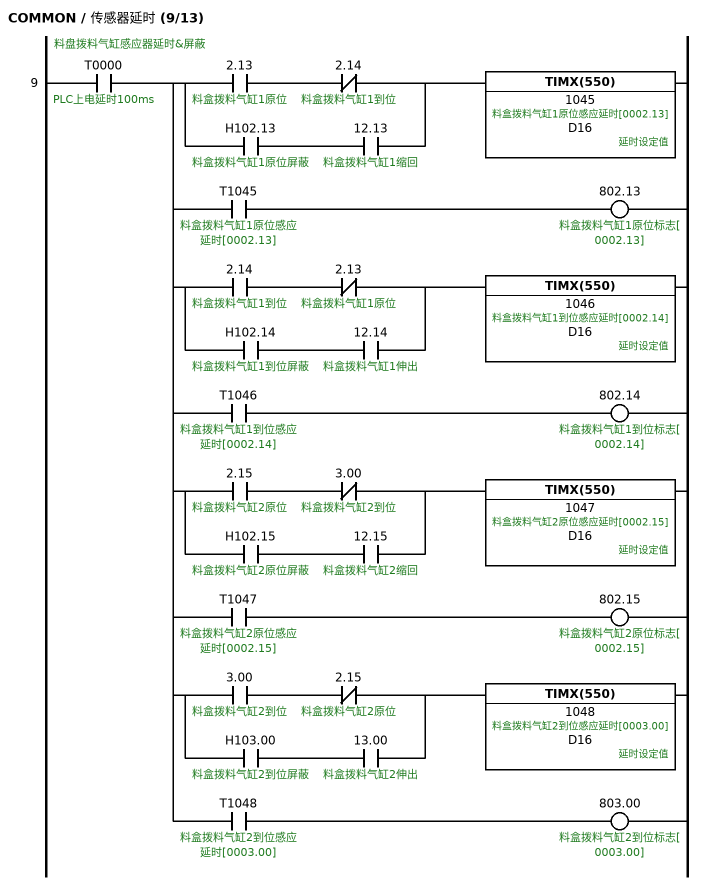
; rung 9: 料盘拨料气缸感应器延时&屏蔽
LD T0000  ; PLC上电延时100ms
OUT TR0
LD 2.13  ; 料盒拨料气缸1原位
ANDNOT 2.14  ; 料盒拨料气缸1到位
LD H102.13  ; 料盒拨料气缸1原位屏蔽
AND 12.13  ; 料盒拨料气缸1缩回
ORLD
ANDLD
TIMX(550) 1045 D16  ; 延时设定值, 料盒拨料气缸1原位感应延时[0002.13]
LD TR0
AND T1045  ; 料盒拨料气缸1原位感应延时[0002.13]
OUT 802.13  ; 料盒拨料气缸1原位标志[0002.13]
LD TR0
LD 2.14  ; 料盒拨料气缸1到位
ANDNOT 2.13  ; 料盒拨料气缸1原位
LD H102.14  ; 料盒拨料气缸1到位屏蔽
AND 12.14  ; 料盒拨料气缸1伸出
ORLD
ANDLD
TIMX(550) 1046 D16  ; 延时设定值, 料盒拨料气缸1到位感应延时[0002.14]
LD TR0
AND T1046  ; 料盒拨料气缸1到位感应延时[0002.14]
OUT 802.14  ; 料盒拨料气缸1到位标志[0002.14]
LD TR0
LD 2.15  ; 料盒拨料气缸2原位
ANDNOT 3.00  ; 料盒拨料气缸2到位
LD H102.15  ; 料盒拨料气缸2原位屏蔽
AND 12.15  ; 料盒拨料气缸2缩回
ORLD
ANDLD
TIMX(550) 1047 D16  ; 延时设定值, 料盒拨料气缸2原位感应延时[0002.15]
LD TR0
AND T1047  ; 料盒拨料气缸2原位感应延时[0002.15]
OUT 802.15  ; 料盒拨料气缸2原位标志[0002.15]
LD TR0
LD 3.00  ; 料盒拨料气缸2到位
ANDNOT 2.15  ; 料盒拨料气缸2原位
LD H103.00  ; 料盒拨料气缸2到位屏蔽
AND 13.00  ; 料盒拨料气缸2伸出
ORLD
ANDLD
TIMX(550) 1048 D16  ; 延时设定值, 料盒拨料气缸2到位感应延时[0003.00]
LD TR0
AND T1048  ; 料盒拨料气缸2到位感应延时[0003.00]
OUT 803.00  ; 料盒拨料气缸2到位标志[0003.00]

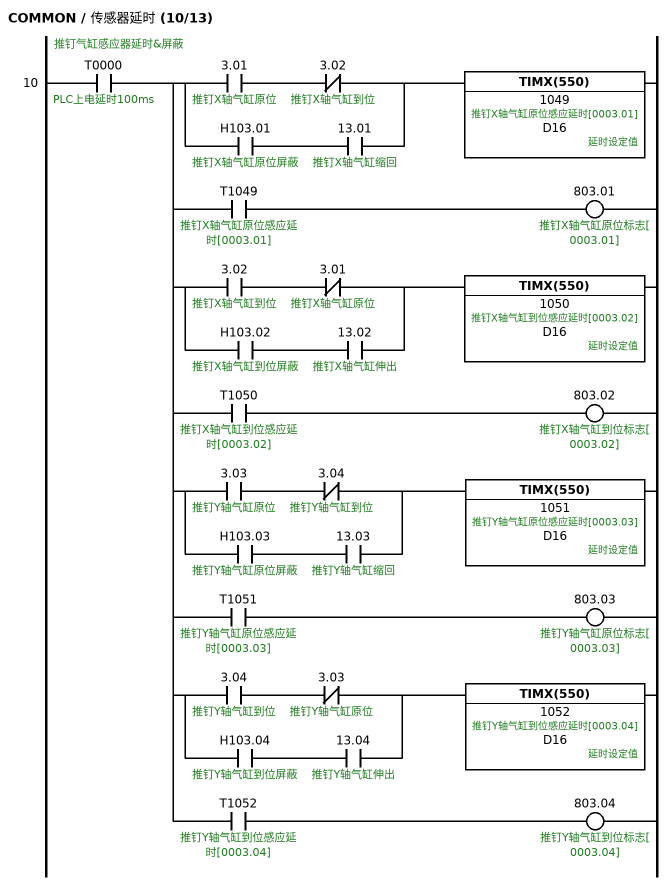
; rung 10: 推钉气缸感应器延时&屏蔽
LD T0000  ; PLC上电延时100ms
OUT TR0
LD 3.01  ; 推钉X轴气缸原位
ANDNOT 3.02  ; 推钉X轴气缸到位
LD H103.01  ; 推钉X轴气缸原位屏蔽
AND 13.01  ; 推钉X轴气缸缩回
ORLD
ANDLD
TIMX(550) 1049 D16  ; 延时设定值, 推钉X轴气缸原位感应延时[0003.01]
LD TR0
AND T1049  ; 推钉X轴气缸原位感应延时[0003.01]
OUT 803.01  ; 推钉X轴气缸原位标志[0003.01]
LD TR0
LD 3.02  ; 推钉X轴气缸到位
ANDNOT 3.01  ; 推钉X轴气缸原位
LD H103.02  ; 推钉X轴气缸到位屏蔽
AND 13.02  ; 推钉X轴气缸伸出
ORLD
ANDLD
TIMX(550) 1050 D16  ; 延时设定值, 推钉X轴气缸到位感应延时[0003.02]
LD TR0
AND T1050  ; 推钉X轴气缸到位感应延时[0003.02]
OUT 803.02  ; 推钉X轴气缸到位标志[0003.02]
LD TR0
LD 3.03  ; 推钉Y轴气缸原位
ANDNOT 3.04  ; 推钉Y轴气缸到位
LD H103.03  ; 推钉Y轴气缸原位屏蔽
AND 13.03  ; 推钉Y轴气缸缩回
ORLD
ANDLD
TIMX(550) 1051 D16  ; 延时设定值, 推钉Y轴气缸原位感应延时[0003.03]
LD TR0
AND T1051  ; 推钉Y轴气缸原位感应延时[0003.03]
OUT 803.03  ; 推钉Y轴气缸原位标志[0003.03]
LD TR0
LD 3.04  ; 推钉Y轴气缸到位
ANDNOT 3.03  ; 推钉Y轴气缸原位
LD H103.04  ; 推钉Y轴气缸到位屏蔽
AND 13.04  ; 推钉Y轴气缸伸出
ORLD
ANDLD
TIMX(550) 1052 D16  ; 延时设定值, 推钉Y轴气缸到位感应延时[0003.04]
LD TR0
AND T1052  ; 推钉Y轴气缸到位感应延时[0003.04]
OUT 803.04  ; 推钉Y轴气缸到位标志[0003.04]

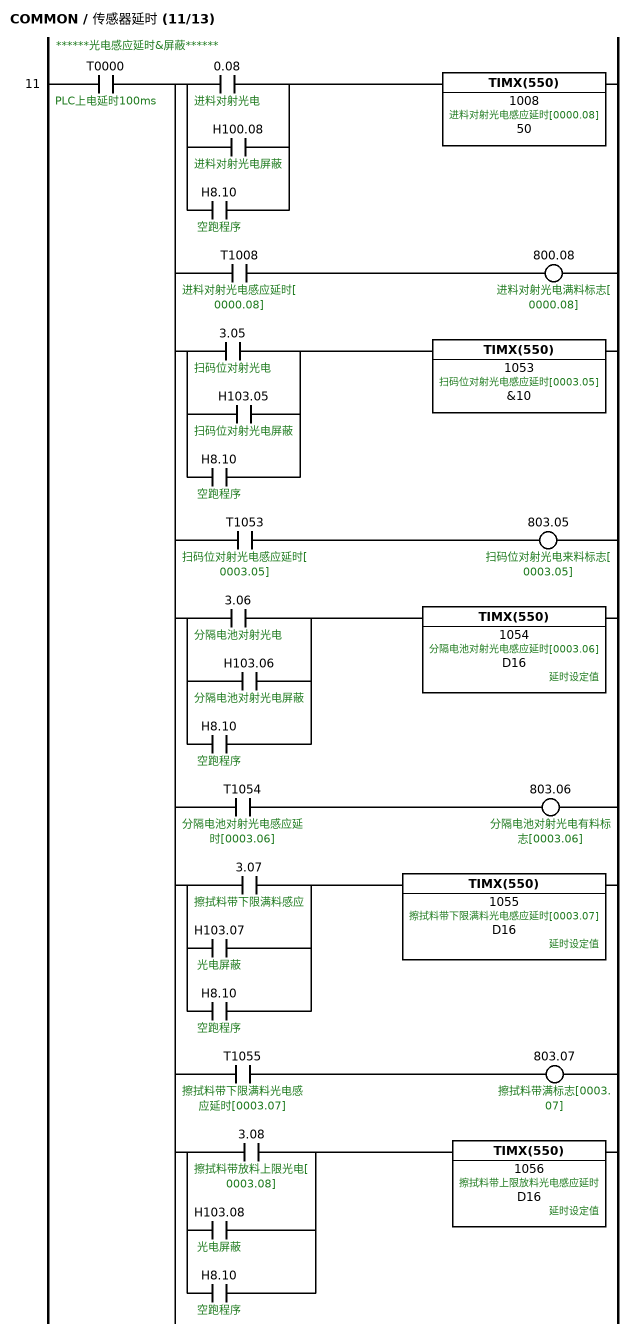

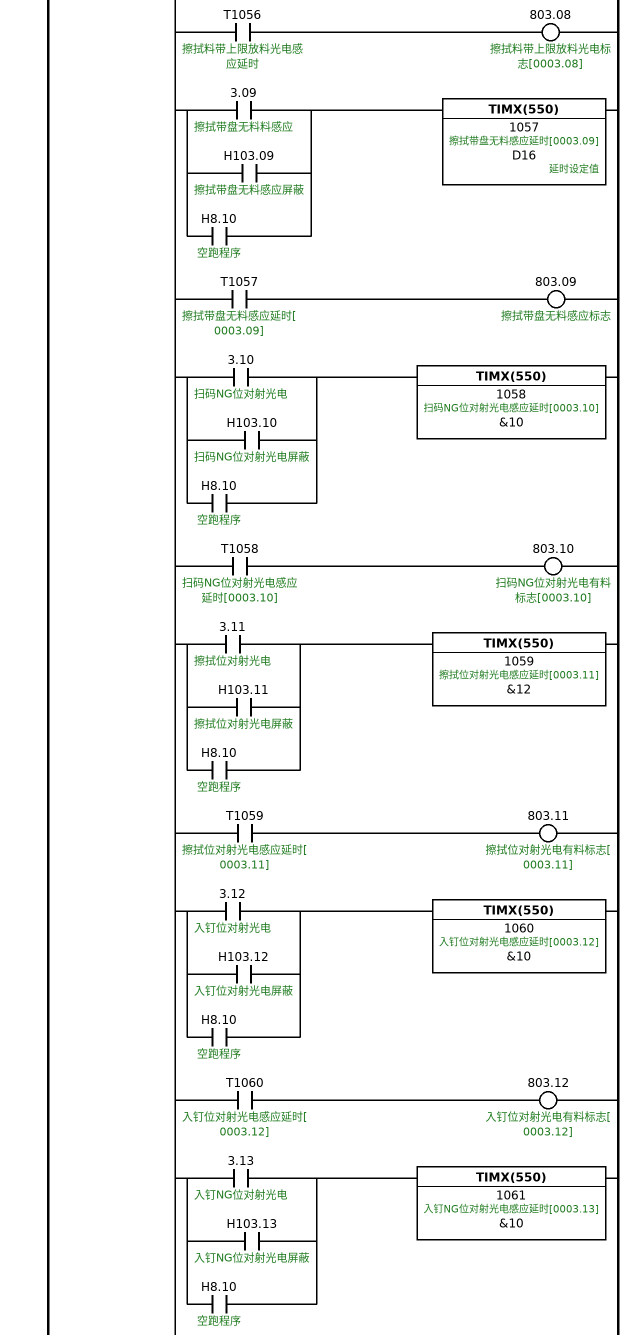

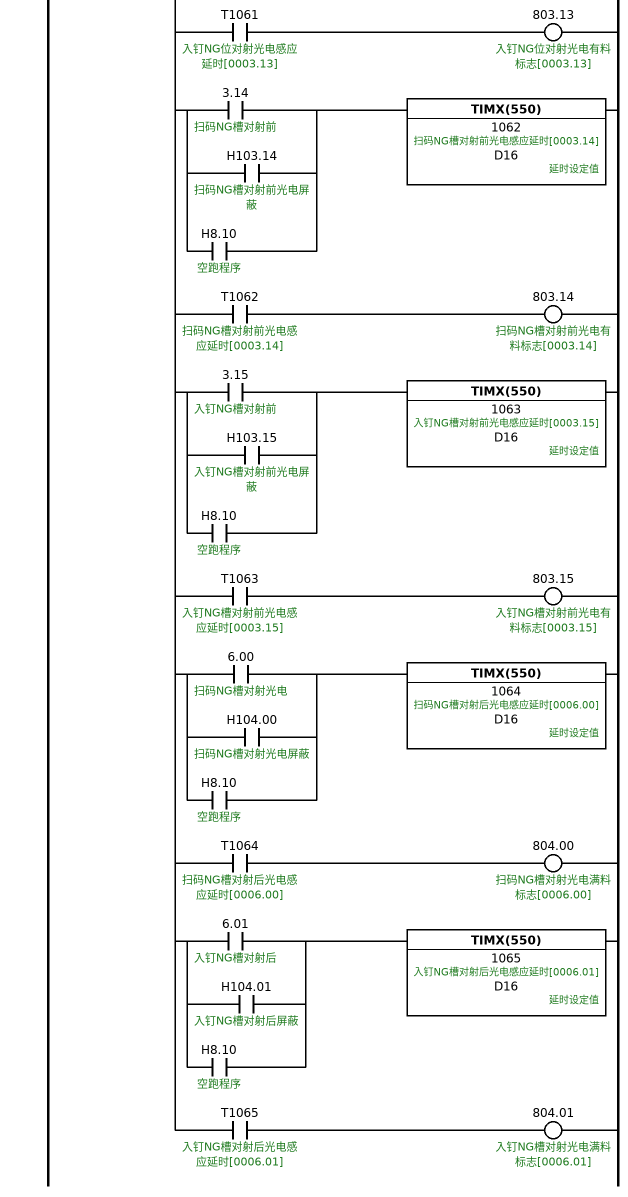
; rung 11: ******光电感应延时&屏蔽******
LD T0000  ; PLC上电延时100ms
OUT TR0
LD 0.08  ; 进料对射光电
OR H100.08  ; 进料对射光电屏蔽
OR H8.10  ; 空跑程序
ANDLD
TIMX(550) 1008 50  ; 进料对射光电感应延时[0000.08]
LD TR0
AND T1008  ; 进料对射光电感应延时[0000.08]
OUT 800.08  ; 进料对射光电满料标志[0000.08]
LD TR0
LD 3.05  ; 扫码位对射光电
OR H103.05  ; 扫码位对射光电屏蔽
OR H8.10  ; 空跑程序
ANDLD
TIMX(550) 1053 &10  ; 扫码位对射光电感应延时[0003.05]
LD TR0
AND T1053  ; 扫码位对射光电感应延时[0003.05]
OUT 803.05  ; 扫码位对射光电来料标志[0003.05]
LD TR0
LD 3.06  ; 分隔电池对射光电
OR H103.06  ; 分隔电池对射光电屏蔽
OR H8.10  ; 空跑程序
ANDLD
TIMX(550) 1054 D16  ; 延时设定值, 分隔电池对射光电感应延时[0003.06]
LD TR0
AND T1054  ; 分隔电池对射光电感应延时[0003.06]
OUT 803.06  ; 分隔电池对射光电有料标志[0003.06]
LD TR0
LD 3.07  ; 擦拭料带下限满料感应
OR H103.07  ; 光电屏蔽
OR H8.10  ; 空跑程序
ANDLD
TIMX(550) 1055 D16  ; 延时设定值, 擦拭料带下限满料光电感应延时[0003.07]
LD TR0
AND T1055  ; 擦拭料带下限满料光电感应延时[0003.07]
OUT 803.07  ; 擦拭料带满标志[0003.07]
LD TR0
LD 3.08  ; 擦拭料带放料上限光电[0003.08]
OR H103.08  ; 光电屏蔽
OR H8.10  ; 空跑程序
ANDLD
TIMX(550) 1056 D16  ; 延时设定值, 擦拭料带上限放料光电感应延时
LD TR0
AND T1056  ; 擦拭料带上限放料光电感应延时
OUT 803.08  ; 擦拭料带上限放料光电标志[0003.08]
LD TR0
LD 3.09  ; 擦拭带盘无料料感应
OR H103.09  ; 擦拭带盘无料感应屏蔽
OR H8.10  ; 空跑程序
ANDLD
TIMX(550) 1057 D16  ; 延时设定值, 擦拭带盘无料感应延时[0003.09]
LD TR0
AND T1057  ; 擦拭带盘无料感应延时[0003.09]
OUT 803.09  ; 擦拭带盘无料感应标志
LD TR0
LD 3.10  ; 扫码NG位对射光电
OR H103.10  ; 扫码NG位对射光电屏蔽
OR H8.10  ; 空跑程序
ANDLD
TIMX(550) 1058 &10  ; 扫码NG位对射光电感应延时[0003.10]
LD TR0
AND T1058  ; 扫码NG位对射光电感应延时[0003.10]
OUT 803.10  ; 扫码NG位对射光电有料标志[0003.10]
LD TR0
LD 3.11  ; 擦拭位对射光电
OR H103.11  ; 擦拭位对射光电屏蔽
OR H8.10  ; 空跑程序
ANDLD
TIMX(550) 1059 &12  ; 擦拭位对射光电感应延时[0003.11]
LD TR0
AND T1059  ; 擦拭位对射光电感应延时[0003.11]
OUT 803.11  ; 擦拭位对射光电有料标志[0003.11]
LD TR0
LD 3.12  ; 入钉位对射光电
OR H103.12  ; 入钉位对射光电屏蔽
OR H8.10  ; 空跑程序
ANDLD
TIMX(550) 1060 &10  ; 入钉位对射光电感应延时[0003.12]
LD TR0
AND T1060  ; 入钉位对射光电感应延时[0003.12]
OUT 803.12  ; 入钉位对射光电有料标志[0003.12]
LD TR0
LD 3.13  ; 入钉NG位对射光电
OR H103.13  ; 入钉NG位对射光电屏蔽
OR H8.10  ; 空跑程序
ANDLD
TIMX(550) 1061 &10  ; 入钉NG位对射光电感应延时[0003.13]
LD TR0
AND T1061  ; 入钉NG位对射光电感应延时[0003.13]
OUT 803.13  ; 入钉NG位对射光电有料标志[0003.13]
LD TR0
LD 3.14  ; 扫码NG槽对射前
OR H103.14  ; 扫码NG槽对射前光电屏蔽
OR H8.10  ; 空跑程序
ANDLD
TIMX(550) 1062 D16  ; 延时设定值, 扫码NG槽对射前光电感应延时[0003.14]
LD TR0
AND T1062  ; 扫码NG槽对射前光电感应延时[0003.14]
OUT 803.14  ; 扫码NG槽对射前光电有料标志[0003.14]
LD TR0
LD 3.15  ; 入钉NG槽对射前
OR H103.15  ; 入钉NG槽对射前光电屏蔽
OR H8.10  ; 空跑程序
ANDLD
TIMX(550) 1063 D16  ; 延时设定值, 入钉NG槽对射前光电感应延时[0003.15]
LD TR0
AND T1063  ; 入钉NG槽对射前光电感应延时[0003.15]
OUT 803.15  ; 入钉NG槽对射前光电有料标志[0003.15]
LD TR0
LD 6.00  ; 扫码NG槽对射光电
OR H104.00  ; 扫码NG槽对射光电屏蔽
OR H8.10  ; 空跑程序
ANDLD
TIMX(550) 1064 D16  ; 延时设定值, 扫码NG槽对射后光电感应延时[0006.00]
LD TR0
AND T1064  ; 扫码NG槽对射后光电感应延时[0006.00]
OUT 804.00  ; 扫码NG槽对射光电满料标志[0006.00]
LD TR0
LD 6.01  ; 入钉NG槽对射后
OR H104.01  ; 入钉NG槽对射后屏蔽
OR H8.10  ; 空跑程序
ANDLD
TIMX(550) 1065 D16  ; 延时设定值, 入钉NG槽对射后光电感应延时[0006.01]
LD TR0
AND T1065  ; 入钉NG槽对射后光电感应延时[0006.01]
OUT 804.01  ; 入钉NG槽对射光电满料标志[0006.01]

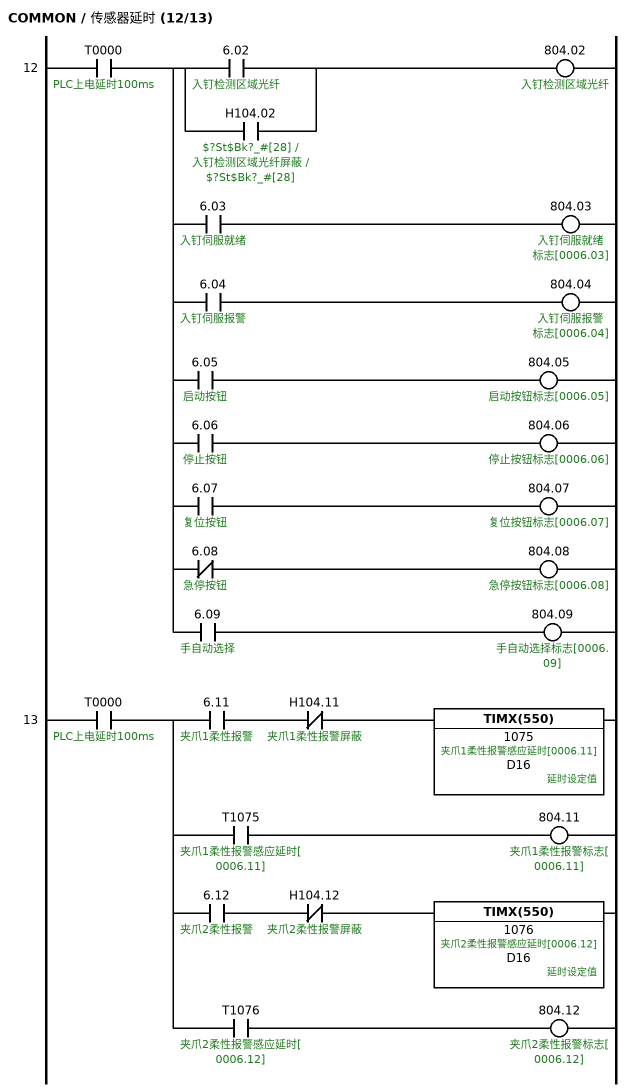
; rung 12
LD T0000  ; PLC上电延时100ms
OUT TR0
LD 6.02  ; 入钉检测区域光纤
OR H104.02  ; $?St$Bk?_#[28] / 入钉检测区域光纤屏蔽 / $?St$Bk?_#[28]
ANDLD
OUT 804.02  ; 入钉检测区域光纤
LD TR0
AND 6.03  ; 入钉伺服就绪
OUT 804.03  ; 入钉伺服就绪 标志[0006.03]
LD TR0
AND 6.04  ; 入钉伺服报警
OUT 804.04  ; 入钉伺服报警 标志[0006.04]
LD TR0
AND 6.05  ; 启动按钮
OUT 804.05  ; 启动按钮标志[0006.05]
LD TR0
AND 6.06  ; 停止按钮
OUT 804.06  ; 停止按钮标志[0006.06]
LD TR0
AND 6.07  ; 复位按钮
OUT 804.07  ; 复位按钮标志[0006.07]
LD TR0
ANDNOT 6.08  ; 急停按钮
OUT 804.08  ; 急停按钮标志[0006.08]
LD TR0
AND 6.09  ; 手自动选择
OUT 804.09  ; 手自动选择标志[0006.09]
; rung 13
LD T0000  ; PLC上电延时100ms
OUT TR0
AND 6.11  ; 夹爪1柔性报警
ANDNOT H104.11  ; 夹爪1柔性报警屏蔽
TIMX(550) 1075 D16  ; 延时设定值, 夹爪1柔性报警感应延时[0006.11]
LD TR0
AND T1075  ; 夹爪1柔性报警感应延时[0006.11]
OUT 804.11  ; 夹爪1柔性报警标志[0006.11]
LD TR0
AND 6.12  ; 夹爪2柔性报警
ANDNOT H104.12  ; 夹爪2柔性报警屏蔽
TIMX(550) 1076 D16  ; 延时设定值, 夹爪2柔性报警感应延时[0006.12]
LD TR0
AND T1076  ; 夹爪2柔性报警感应延时[0006.12]
OUT 804.12  ; 夹爪2柔性报警标志[0006.12]

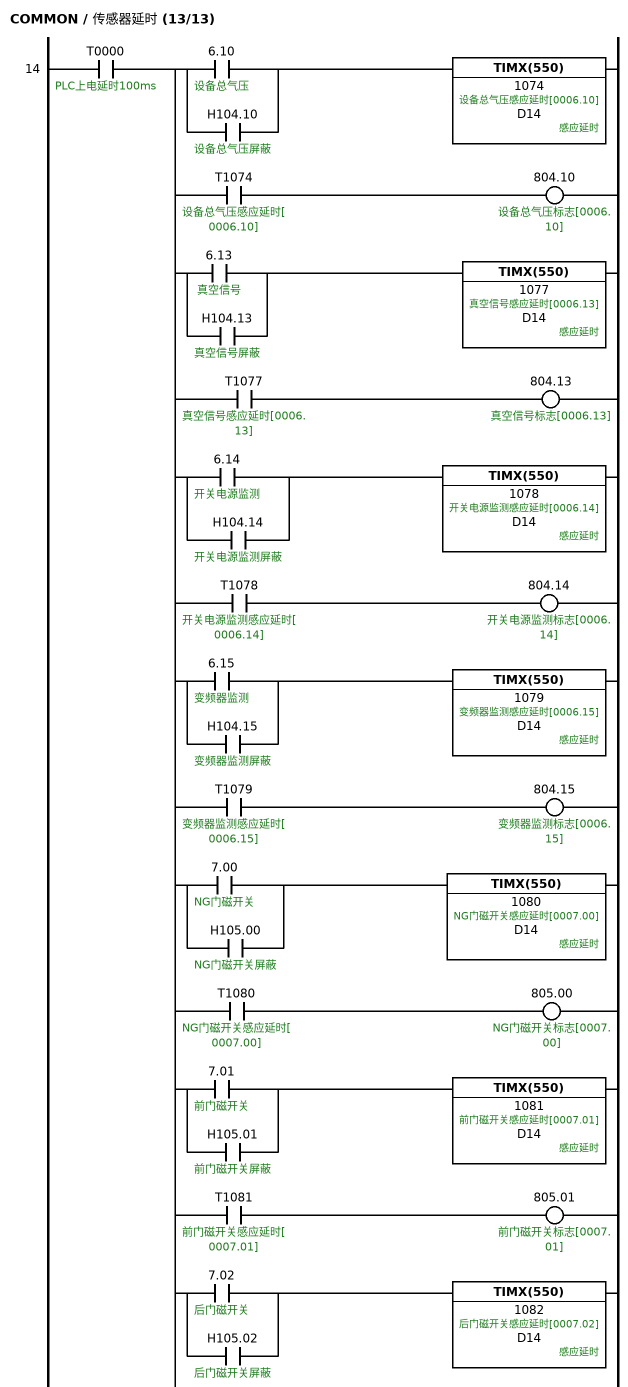

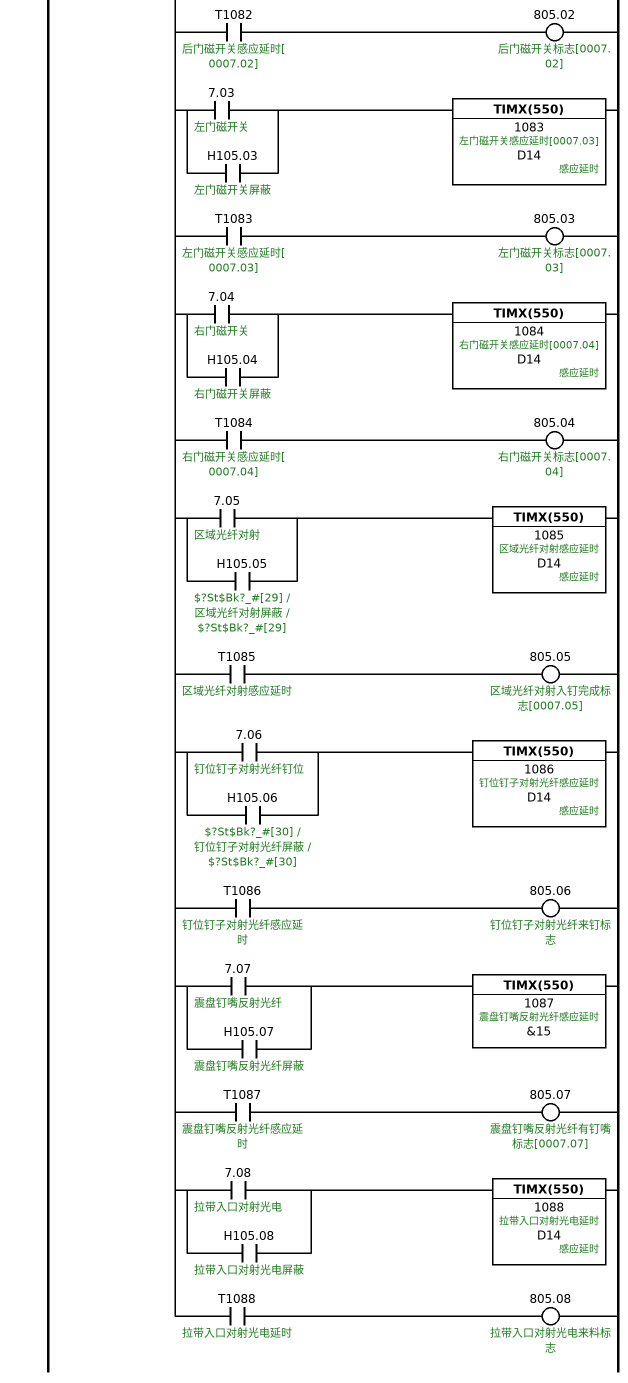
; rung 14
LD T0000  ; PLC上电延时100ms
OUT TR0
LD 6.10  ; 设备总气压
OR H104.10  ; 设备总气压屏蔽
ANDLD
TIMX(550) 1074 D14  ; 感应延时, 设备总气压感应延时[0006.10]
LD TR0
AND T1074  ; 设备总气压感应延时[0006.10]
OUT 804.10  ; 设备总气压标志[0006.10]
LD TR0
LD 6.13  ; 真空信号
OR H104.13  ; 真空信号屏蔽
ANDLD
TIMX(550) 1077 D14  ; 感应延时, 真空信号感应延时[0006.13]
LD TR0
AND T1077  ; 真空信号感应延时[0006.13]
OUT 804.13  ; 真空信号标志[0006.13]
LD TR0
LD 6.14  ; 开关电源监测
OR H104.14  ; 开关电源监测屏蔽
ANDLD
TIMX(550) 1078 D14  ; 感应延时, 开关电源监测感应延时[0006.14]
LD TR0
AND T1078  ; 开关电源监测感应延时[0006.14]
OUT 804.14  ; 开关电源监测标志[0006.14]
LD TR0
LD 6.15  ; 变频器监测
OR H104.15  ; 变频器监测屏蔽
ANDLD
TIMX(550) 1079 D14  ; 感应延时, 变频器监测感应延时[0006.15]
LD TR0
AND T1079  ; 变频器监测感应延时[0006.15]
OUT 804.15  ; 变频器监测标志[0006.15]
LD TR0
LD 7.00  ; NG门磁开关
OR H105.00  ; NG门磁开关屏蔽
ANDLD
TIMX(550) 1080 D14  ; 感应延时, NG门磁开关感应延时[0007.00]
LD TR0
AND T1080  ; NG门磁开关感应延时[0007.00]
OUT 805.00  ; NG门磁开关标志[0007.00]
LD TR0
LD 7.01  ; 前门磁开关
OR H105.01  ; 前门磁开关屏蔽
ANDLD
TIMX(550) 1081 D14  ; 感应延时, 前门磁开关感应延时[0007.01]
LD TR0
AND T1081  ; 前门磁开关感应延时[0007.01]
OUT 805.01  ; 前门磁开关标志[0007.01]
LD TR0
LD 7.02  ; 后门磁开关
OR H105.02  ; 后门磁开关屏蔽
ANDLD
TIMX(550) 1082 D14  ; 感应延时, 后门磁开关感应延时[0007.02]
LD TR0
AND T1082  ; 后门磁开关感应延时[0007.02]
OUT 805.02  ; 后门磁开关标志[0007.02]
LD TR0
LD 7.03  ; 左门磁开关
OR H105.03  ; 左门磁开关屏蔽
ANDLD
TIMX(550) 1083 D14  ; 感应延时, 左门磁开关感应延时[0007.03]
LD TR0
AND T1083  ; 左门磁开关感应延时[0007.03]
OUT 805.03  ; 左门磁开关标志[0007.03]
LD TR0
LD 7.04  ; 右门磁开关
OR H105.04  ; 右门磁开关屏蔽
ANDLD
TIMX(550) 1084 D14  ; 感应延时, 右门磁开关感应延时[0007.04]
LD TR0
AND T1084  ; 右门磁开关感应延时[0007.04]
OUT 805.04  ; 右门磁开关标志[0007.04]
LD TR0
LD 7.05  ; 区域光纤对射
OR H105.05  ; $?St$Bk?_#[29] / 区域光纤对射屏蔽 / $?St$Bk?_#[29]
ANDLD
TIMX(550) 1085 D14  ; 感应延时, 区域光纤对射感应延时
LD TR0
AND T1085  ; 区域光纤对射感应延时
OUT 805.05  ; 区域光纤对射入钉完成标志[0007.05]
LD TR0
LD 7.06  ; 钉位钉子对射光纤钉位
OR H105.06  ; $?St$Bk?_#[30] / 钉位钉子对射光纤屏蔽 / $?St$Bk?_#[30]
ANDLD
TIMX(550) 1086 D14  ; 感应延时, 钉位钉子对射光纤感应延时
LD TR0
AND T1086  ; 钉位钉子对射光纤感应延时
OUT 805.06  ; 钉位钉子对射光纤来钉标志
LD TR0
LD 7.07  ; 震盘钉嘴反射光纤
OR H105.07  ; 震盘钉嘴反射光纤屏蔽
ANDLD
TIMX(550) 1087 &15  ; 震盘钉嘴反射光纤感应延时
LD TR0
AND T1087  ; 震盘钉嘴反射光纤感应延时
OUT 805.07  ; 震盘钉嘴反射光纤有钉嘴标志[0007.07]
LD TR0
LD 7.08  ; 拉带入口对射光电
OR H105.08  ; 拉带入口对射光电屏蔽
ANDLD
TIMX(550) 1088 D14  ; 感应延时, 拉带入口对射光电延时
LD TR0
AND T1088  ; 拉带入口对射光电延时
OUT 805.08  ; 拉带入口对射光电来料标志

### Section 动作延时

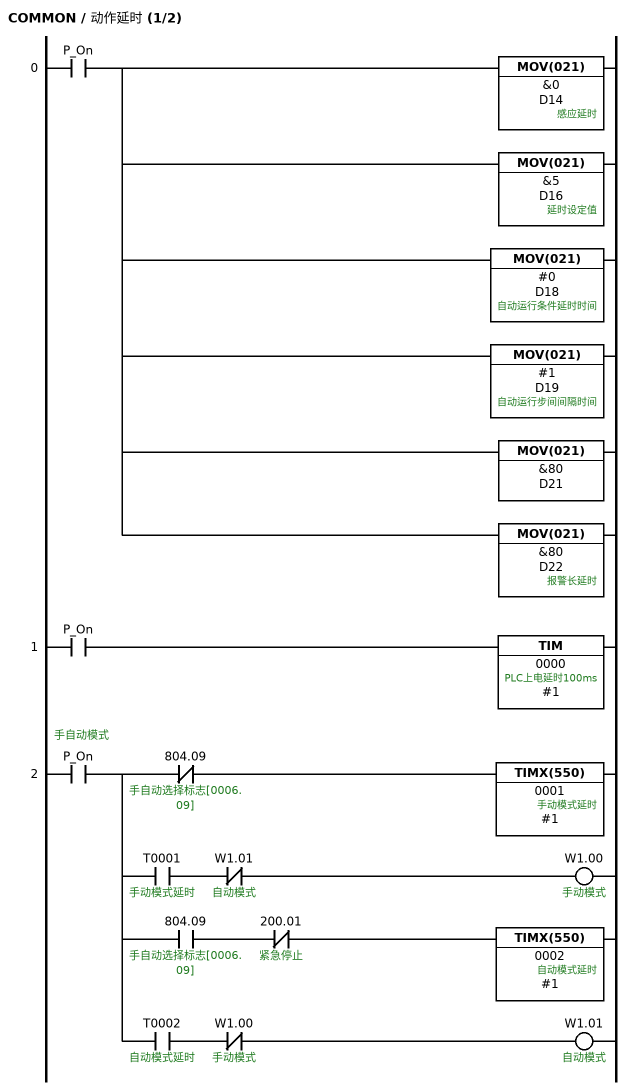
; rung 0
LD P_On
MOV(021) &0 D14  ; 感应延时
MOV(021) &5 D16  ; 延时设定值
MOV(021) #0 D18  ; 自动运行条件延时时间
MOV(021) #1 D19  ; 自动运行步间间隔时间
MOV(021) &80 D21
MOV(021) &80 D22  ; 报警长延时
; rung 1
LD P_On
TIM 0000 #1  ; PLC上电延时100ms
; rung 2: 手自动模式
LD P_On
OUT TR0
ANDNOT 804.09  ; 手自动选择标志[0006.09]
TIMX(550) 0001 #1  ; 手动模式延时
LD TR0
AND T0001  ; 手动模式延时
ANDNOT W1.01  ; 自动模式
OUT W1.00  ; 手动模式
LD TR0
AND 804.09  ; 手自动选择标志[0006.09]
ANDNOT 200.01  ; 紧急停止
TIMX(550) 0002 #1  ; 自动模式延时
LD TR0
AND T0002  ; 自动模式延时
ANDNOT W1.00  ; 手动模式
OUT W1.01  ; 自动模式

